LIN {X 53.277,Y 73.918,Z 73.500,A 180.000,B 0.000,C 180.000} C_DIS
LIN {X 53.455,Y 73.864,Z 73.500,A 180.000,B 0.000,C 180.000} C_DIS
LIN {X 75.444,Y 66.446,Z 73.500,A 180.000,B 0.000,C 180.000} C_DIS
LIN {X 75.534,Y 66.414,Z 73.500,A 180.000,B 0.000,C 180.000} C_DIS
LIN {X 75.623,Y 66.379,Z 73.500,A 180.000,B 0.000,C 180.000} C_DIS
LIN {X 75.739,Y 66.327,Z 73.500,A 180.000,B 0.000,C 180.000} C_DIS
LIN {X 75.802,Y 66.296,Z 73.500,A 180.000,B 0.000,C 180.000} C_DIS
LIN {X 75.891,Y 66.247,Z 73.500,A 180.000,B 0.000,C 180.000} C_DIS
LIN {X 75.980,Y 66.194,Z 73.500,A 180.000,B 0.000,C 180.000} C_DIS
LIN {X 76.052,Y 66.148,Z 73.500,A 180.000,B 0.000,C 180.000} C_DIS
LIN {X 76.159,Y 66.072,Z 73.500,A 180.000,B 0.000,C 180.000} C_DIS
LIN {X 76.223,Y 66.022,Z 73.500,A 180.000,B 0.000,C 180.000} C_DIS
LIN {X 76.287,Y 65.969,Z 73.500,A 180.000,B 0.000,C 180.000} C_DIS
LIN {X 76.338,Y 65.924,Z 73.500,A 180.000,B 0.000,C 180.000} C_DIS
LIN {X 76.406,Y 65.860,Z 73.500,A 180.000,B 0.000,C 180.000} C_DIS
LIN {X 76.474,Y 65.791,Z 73.500,A 180.000,B 0.000,C 180.000} C_DIS
LIN {X 76.517,Y 65.744,Z 73.500,A 180.000,B 0.000,C 180.000} C_DIS
LIN {X 76.628,Y 65.612,Z 73.500,A 180.000,B 0.000,C 180.000} C_DIS
LIN {X 76.696,Y 65.521,Z 73.500,A 180.000,B 0.000,C 180.000} C_DIS
LIN {X 76.755,Y 65.433,Z 73.500,A 180.000,B 0.000,C 180.000} C_DIS
LIN {X 76.861,Y 65.254,Z 73.500,A 180.000,B 0.000,C 180.000} C_DIS
LIN {X 76.874,Y 65.229,Z 73.500,A 180.000,B 0.000,C 180.000} C_DIS
LIN {X 76.948,Y 65.075,Z 73.500,A 180.000,B 0.000,C 180.000} C_DIS
LIN {X 77.018,Y 64.897,Z 73.500,A 180.000,B 0.000,C 180.000} C_DIS
LIN {X 77.053,Y 64.789,Z 73.500,A 180.000,B 0.000,C 180.000} C_DIS
LIN {X 77.073,Y 64.718,Z 73.500,A 180.000,B 0.000,C 180.000} C_DIS
LIN {X 77.114,Y 64.539,Z 73.500,A 180.000,B 0.000,C 180.000} C_DIS
LIN {X 77.141,Y 64.360,Z 73.500,A 180.000,B 0.000,C 180.000} C_DIS
LIN {X 77.155,Y 64.182,Z 73.500,A 180.000,B 0.000,C 180.000} C_DIS
LIN {X 77.157,Y 64.003,Z 73.500,A 180.000,B 0.000,C 180.000} C_DIS
LIN {X 77.145,Y 63.824,Z 73.500,A 180.000,B 0.000,C 180.000} C_DIS
LIN {X 77.121,Y 63.645,Z 73.500,A 180.000,B 0.000,C 180.000} C_DIS
LIN {X 77.083,Y 63.467,Z 73.500,A 180.000,B 0.000,C 180.000} C_DIS
LIN {X 77.053,Y 63.357,Z 73.500,A 180.000,B 0.000,C 180.000} C_DIS
LIN {X 77.031,Y 63.288,Z 73.500,A 180.000,B 0.000,C 180.000} C_DIS
LIN {X 76.971,Y 63.109,Z 73.500,A 180.000,B 0.000,C 180.000} C_DIS
LIN {X 70.639,Y 44.338,Z 73.500,A 180.000,B 0.000,C 180.000} C_DIS
LIN {X 70.617,Y 44.276,Z 73.500,A 180.000,B 0.000,C 180.000} C_DIS
LIN {X 70.572,Y 44.159,Z 73.500,A 180.000,B 0.000,C 180.000} C_DIS
LIN {X 70.489,Y 43.981,Z 73.500,A 180.000,B 0.000,C 180.000} C_DIS
LIN {X 70.439,Y 43.887,Z 73.500,A 180.000,B 0.000,C 180.000} C_DIS
LIN {X 70.388,Y 43.802,Z 73.500,A 180.000,B 0.000,C 180.000} C_DIS
LIN {X 70.266,Y 43.623,Z 73.500,A 180.000,B 0.000,C 180.000} C_DIS
LIN {X 70.260,Y 43.615,Z 73.500,A 180.000,B 0.000,C 180.000} C_DIS
LIN {X 70.118,Y 43.444,Z 73.500,A 180.000,B 0.000,C 180.000} C_DIS
LIN {X 70.081,Y 43.404,Z 73.500,A 180.000,B 0.000,C 180.000} C_DIS
LIN {X 69.939,Y 43.266,Z 73.500,A 180.000,B 0.000,C 180.000} C_DIS
LIN {X 69.902,Y 43.233,Z 73.500,A 180.000,B 0.000,C 180.000} C_DIS
LIN {X 69.724,Y 43.092,Z 73.500,A 180.000,B 0.000,C 180.000} C_DIS
LIN {X 69.717,Y 43.087,Z 73.500,A 180.000,B 0.000,C 180.000} C_DIS
LIN {X 69.545,Y 42.975,Z 73.500,A 180.000,B 0.000,C 180.000} C_DIS
LIN {X 69.426,Y 42.908,Z 73.500,A 180.000,B 0.000,C 180.000} C_DIS
LIN {X 69.366,Y 42.878,Z 73.500,A 180.000,B 0.000,C 180.000} C_DIS
LIN {X 69.187,Y 42.798,Z 73.500,A 180.000,B 0.000,C 180.000} C_DIS
LIN {X 69.008,Y 42.735,Z 73.500,A 180.000,B 0.000,C 180.000} C_DIS
LIN {X 68.989,Y 42.729,Z 73.500,A 180.000,B 0.000,C 180.000} C_DIS
LIN {X 68.830,Y 42.687,Z 73.500,A 180.000,B 0.000,C 180.000} C_DIS
LIN {X 68.651,Y 42.652,Z 73.500,A 180.000,B 0.000,C 180.000} C_DIS
LIN {X 68.562,Y 42.640,Z 73.500,A 180.000,B 0.000,C 180.000} C_DIS
LIN {X 68.472,Y 42.631,Z 73.500,A 180.000,B 0.000,C 180.000} C_DIS
LIN {X 68.383,Y 42.625,Z 73.500,A 180.000,B 0.000,C 180.000} C_DIS
LIN {X 68.293,Y 42.622,Z 73.500,A 180.000,B 0.000,C 180.000} C_DIS
LIN {X 68.204,Y 42.623,Z 73.500,A 180.000,B 0.000,C 180.000} C_DIS
LIN {X 68.115,Y 42.627,Z 73.500,A 180.000,B 0.000,C 180.000} C_DIS
LIN {X 68.025,Y 42.634,Z 73.500,A 180.000,B 0.000,C 180.000} C_DIS
LIN {X 67.936,Y 42.644,Z 73.500,A 180.000,B 0.000,C 180.000} C_DIS
LIN {X 67.846,Y 42.657,Z 73.500,A 180.000,B 0.000,C 180.000} C_DIS
LIN {X 67.757,Y 42.674,Z 73.500,A 180.000,B 0.000,C 180.000} C_DIS
LIN {X 67.668,Y 42.694,Z 73.500,A 180.000,B 0.000,C 180.000} C_DIS
LIN {X 67.578,Y 42.718,Z 73.500,A 180.000,B 0.000,C 180.000} C_DIS
LIN {X 67.541,Y 42.729,Z 73.500,A 180.000,B 0.000,C 180.000} C_DIS
LIN {X 67.399,Y 42.776,Z 73.500,A 180.000,B 0.000,C 180.000} C_DIS
LIN {X 47.482,Y 49.495,Z 73.500,A 180.000,B 0.000,C 180.000} C_DIS
; Link Move Starts
LIN {X 47.184,Y 49.595,Z 73.500,A 180.000,B 0.000,C 180.000} C_DIS
LIN {X 46.885,Y 49.696,Z 73.499,A 180.000,B 0.000,C 180.000} C_DIS
LIN {X 46.587,Y 49.797,Z 73.498,A 180.000,B 0.000,C 180.000} C_DIS
LIN {X 46.288,Y 49.897,Z 73.496,A 180.000,B 0.000,C 180.000} C_DIS
LIN {X 45.990,Y 49.998,Z 73.494,A 180.000,B 0.000,C 180.000} C_DIS
LIN {X 45.692,Y 50.099,Z 73.491,A 180.000,B 0.000,C 180.000} C_DIS
LIN {X 45.393,Y 50.200,Z 73.488,A 180.000,B 0.000,C 180.000} C_DIS
LIN {X 45.247,Y 50.259,Z 73.487,A 180.000,B 0.000,C 180.000} C_DIS
LIN {X 45.105,Y 50.326,Z 73.485,A 180.000,B 0.000,C 180.000} C_DIS
LIN {X 44.967,Y 50.403,Z 73.483,A 180.000,B 0.000,C 180.000} C_DIS
LIN {X 44.834,Y 50.487,Z 73.481,A 180.000,B 0.000,C 180.000} C_DIS
LIN {X 44.707,Y 50.581,Z 73.479,A 180.000,B 0.000,C 180.000} C_DIS
LIN {X 44.587,Y 50.682,Z 73.477,A 180.000,B 0.000,C 180.000} C_DIS
LIN {X 44.472,Y 50.790,Z 73.474,A 180.000,B 0.000,C 180.000} C_DIS
LIN {X 44.365,Y 50.905,Z 73.472,A 180.000,B 0.000,C 180.000} C_DIS
LIN {X 44.265,Y 51.027,Z 73.469,A 180.000,B 0.000,C 180.000} C_DIS
LIN {X 44.173,Y 51.155,Z 73.467,A 180.000,B 0.000,C 180.000} C_DIS
LIN {X 44.090,Y 51.288,Z 73.464,A 180.000,B 0.000,C 180.000} C_DIS
LIN {X 44.014,Y 51.427,Z 73.461,A 180.000,B 0.000,C 180.000} C_DIS
LIN {X 43.948,Y 51.570,Z 73.459,A 180.000,B 0.000,C 180.000} C_DIS
LIN {X 43.891,Y 51.716,Z 73.456,A 180.000,B 0.000,C 180.000} C_DIS
LIN {X 43.843,Y 51.867,Z 73.452,A 180.000,B 0.000,C 180.000} C_DIS
LIN {X 43.805,Y 52.019,Z 73.449,A 180.000,B 0.000,C 180.000} C_DIS
LIN {X 43.777,Y 52.174,Z 73.446,A 180.000,B 0.000,C 180.000} C_DIS
LIN {X 43.758,Y 52.331,Z 73.443,A 180.000,B 0.000,C 180.000} C_DIS
LIN {X 43.749,Y 52.488,Z 73.439,A 180.000,B 0.000,C 180.000} C_DIS
LIN {X 43.750,Y 52.645,Z 73.436,A 180.000,B 0.000,C 180.000} C_DIS
LIN {X 43.761,Y 52.803,Z 73.432,A 180.000,B 0.000,C 180.000} C_DIS
LIN {X 43.782,Y 52.959,Z 73.428,A 180.000,B 0.000,C 180.000} C_DIS
LIN {X 43.813,Y 53.113,Z 73.425,A 180.000,B 0.000,C 180.000} C_DIS
LIN {X 43.853,Y 53.265,Z 73.421,A 180.000,B 0.000,C 180.000} C_DIS
LIN {X 43.902,Y 53.415,Z 73.417,A 180.000,B 0.000,C 180.000} C_DIS
LIN {X 43.952,Y 53.564,Z 73.413,A 180.000,B 0.000,C 180.000} C_DIS
LIN {X 44.003,Y 53.714,Z 73.409,A 180.000,B 0.000,C 180.000} C_DIS
LIN {X 44.053,Y 53.863,Z 73.405,A 180.000,B 0.000,C 180.000} C_DIS
LIN {X 44.103,Y 54.012,Z 73.400,A 180.000,B 0.000,C 180.000} C_DIS
LIN {X 44.154,Y 54.161,Z 73.396,A 180.000,B 0.000,C 180.000} C_DIS
LIN {X 44.204,Y 54.310,Z 73.392,A 180.000,B 0.000,C 180.000} C_DIS
LIN {X 44.254,Y 54.460,Z 73.387,A 180.000,B 0.000,C 180.000} C_DIS
LIN {X 44.305,Y 54.609,Z 73.383,A 180.000,B 0.000,C 180.000} C_DIS
LIN {X 44.355,Y 54.758,Z 73.378,A 180.000,B 0.000,C 180.000} C_DIS
LIN {X 44.405,Y 54.907,Z 73.373,A 180.000,B 0.000,C 180.000} C_DIS
LIN {X 44.456,Y 55.057,Z 73.369,A 180.000,B 0.000,C 180.000} C_DIS
LIN {X 44.506,Y 55.206,Z 73.364,A 180.000,B 0.000,C 180.000} C_DIS
LIN {X 44.556,Y 55.355,Z 73.359,A 180.000,B 0.000,C 180.000} C_DIS
LIN {X 44.607,Y 55.504,Z 73.354,A 180.000,B 0.000,C 180.000} C_DIS
LIN {X 44.632,Y 55.579,Z 73.351,A 180.000,B 0.000,C 180.000} C_DIS
LIN {X 44.657,Y 55.654,Z 73.349,A 180.000,B 0.000,C 180.000} C_DIS
LIN {X 44.682,Y 55.728,Z 73.346,A 180.000,B 0.000,C 180.000} C_DIS
LIN {X 44.707,Y 55.803,Z 73.344,A 180.000,B 0.000,C 180.000} C_DIS
LIN {X 44.733,Y 55.877,Z 73.341,A 180.000,B 0.000,C 180.000} C_DIS
LIN {X 44.758,Y 55.952,Z 73.339,A 180.000,B 0.000,C 180.000} C_DIS
LIN {X 44.783,Y 56.027,Z 73.336,A 180.000,B 0.000,C 180.000} C_DIS
LIN {X 44.833,Y 56.176,Z 73.331,A 180.000,B 0.000,C 180.000} C_DIS
LIN {X 44.884,Y 56.325,Z 73.325,A 180.000,B 0.000,C 180.000} C_DIS
LIN {X 44.934,Y 56.474,Z 73.320,A 180.000,B 0.000,C 180.000} C_DIS
LIN {X 44.984,Y 56.624,Z 73.315,A 180.000,B 0.000,C 180.000} C_DIS
LIN {X 45.035,Y 56.773,Z 73.309,A 180.000,B 0.000,C 180.000} C_DIS
LIN {X 45.060,Y 56.848,Z 73.307,A 180.000,B 0.000,C 180.000} C_DIS
LIN {X 45.110,Y 56.997,Z 73.301,A 180.000,B 0.000,C 180.000} C_DIS
LIN {X 45.186,Y 57.221,Z 73.293,A 180.000,B 0.000,C 180.000} C_DIS
LIN {X 45.236,Y 57.370,Z 73.287,A 180.000,B 0.000,C 180.000} C_DIS
LIN {X 45.261,Y 57.444,Z 73.285,A 180.000,B 0.000,C 180.000} C_DIS
LIN {X 45.312,Y 57.594,Z 73.279,A 180.000,B 0.000,C 180.000} C_DIS
LIN {X 45.387,Y 57.818,Z 73.271,A 180.000,B 0.000,C 180.000} C_DIS
LIN {X 45.437,Y 57.967,Z 73.265,A 180.000,B 0.000,C 180.000} C_DIS
LIN {X 45.463,Y 58.041,Z 73.263,A 180.000,B 0.000,C 180.000} C_DIS
LIN {X 45.513,Y 58.191,Z 73.257,A 180.000,B 0.000,C 180.000} C_DIS
LIN {X 45.588,Y 58.414,Z 73.249,A 180.000,B 0.000,C 180.000} C_DIS
LIN {X 45.639,Y 58.564,Z 73.243,A 180.000,B 0.000,C 180.000} C_DIS
LIN {X 45.664,Y 58.638,Z 73.241,A 180.000,B 0.000,C 180.000} C_DIS
LIN {X 45.714,Y 58.788,Z 73.235,A 180.000,B 0.000,C 180.000} C_DIS
LIN {X 45.790,Y 59.011,Z 73.227,A 180.000,B 0.000,C 180.000} C_DIS
LIN {X 45.840,Y 59.161,Z 73.221,A 180.000,B 0.000,C 180.000} C_DIS
LIN {X 45.865,Y 59.235,Z 73.219,A 180.000,B 0.000,C 180.000} C_DIS
LIN {X 45.916,Y 59.385,Z 73.213,A 180.000,B 0.000,C 180.000} C_DIS
LIN {X 46.067,Y 59.832,Z 73.197,A 180.000,B 0.000,C 180.000} C_DIS
LIN {X 46.117,Y 59.981,Z 73.191,A 180.000,B 0.000,C 180.000} C_DIS
LIN {X 46.268,Y 60.429,Z 73.175,A 180.000,B 0.000,C 180.000} C_DIS
LIN {X 46.318,Y 60.578,Z 73.169,A 180.000,B 0.000,C 180.000} C_DIS
LIN {X 46.495,Y 61.101,Z 73.150,A 180.000,B 0.000,C 180.000} C_DIS
LIN {X 46.646,Y 61.548,Z 73.133,A 180.000,B 0.000,C 180.000} C_DIS
LIN {X 46.696,Y 61.698,Z 73.128,A 180.000,B 0.000,C 180.000} C_DIS
LIN {X 46.847,Y 62.145,Z 73.111,A 180.000,B 0.000,C 180.000} C_DIS
LIN {X 46.897,Y 62.295,Z 73.106,A 180.000,B 0.000,C 180.000} C_DIS
LIN {X 47.149,Y 63.041,Z 73.078,A 180.000,B 0.000,C 180.000} C_DIS
LIN {X 47.275,Y 63.414,Z 73.065,A 180.000,B 0.000,C 180.000} C_DIS
LIN {X 47.426,Y 63.862,Z 73.048,A 180.000,B 0.000,C 180.000} C_DIS
LIN {X 48.005,Y 65.578,Z 72.985,A 180.000,B 0.000,C 180.000} C_DIS
LIN {X 48.962,Y 68.413,Z 72.880,A 180.000,B 0.000,C 180.000} C_DIS
LIN {X 49.012,Y 68.563,Z 72.875,A 180.000,B 0.000,C 180.000} C_DIS
LIN {X 49.163,Y 69.010,Z 72.858,A 180.000,B 0.000,C 180.000} C_DIS
LIN {X 49.213,Y 69.160,Z 72.853,A 180.000,B 0.000,C 180.000} C_DIS
LIN {X 49.364,Y 69.607,Z 72.836,A 180.000,B 0.000,C 180.000} C_DIS
LIN {X 49.390,Y 69.682,Z 72.834,A 180.000,B 0.000,C 180.000} C_DIS
LIN {X 49.440,Y 69.831,Z 72.828,A 180.000,B 0.000,C 180.000} C_DIS
LIN {X 49.591,Y 70.279,Z 72.812,A 180.000,B 0.000,C 180.000} C_DIS
LIN {X 49.641,Y 70.428,Z 72.806,A 180.000,B 0.000,C 180.000} C_DIS
LIN {X 49.792,Y 70.876,Z 72.790,A 180.000,B 0.000,C 180.000} C_DIS
LIN {X 49.843,Y 71.025,Z 72.784,A 180.000,B 0.000,C 180.000} C_DIS
LIN {X 49.918,Y 71.249,Z 72.776,A 180.000,B 0.000,C 180.000} C_DIS
LIN {X 49.968,Y 71.398,Z 72.770,A 180.000,B 0.000,C 180.000} C_DIS
LIN {X 49.994,Y 71.473,Z 72.768,A 180.000,B 0.000,C 180.000} C_DIS
LIN {X 50.044,Y 71.622,Z 72.762,A 180.000,B 0.000,C 180.000} C_DIS
LIN {X 50.120,Y 71.846,Z 72.754,A 180.000,B 0.000,C 180.000} C_DIS
LIN {X 50.170,Y 71.995,Z 72.748,A 180.000,B 0.000,C 180.000} C_DIS
LIN {X 50.195,Y 72.070,Z 72.746,A 180.000,B 0.000,C 180.000} C_DIS
LIN {X 50.245,Y 72.219,Z 72.740,A 180.000,B 0.000,C 180.000} C_DIS
LIN {X 50.271,Y 72.293,Z 72.737,A 180.000,B 0.000,C 180.000} C_DIS
LIN {X 50.297,Y 72.368,Z 72.735,A 180.000,B 0.000,C 180.000} C_DIS
LIN {X 50.325,Y 72.441,Z 72.732,A 180.000,B 0.000,C 180.000} C_DIS
LIN {X 50.356,Y 72.514,Z 72.729,A 180.000,B 0.000,C 180.000} C_DIS
LIN {X 50.389,Y 72.585,Z 72.726,A 180.000,B 0.000,C 180.000} C_DIS
LIN {X 50.424,Y 72.656,Z 72.724,A 180.000,B 0.000,C 180.000} C_DIS
LIN {X 50.462,Y 72.725,Z 72.721,A 180.000,B 0.000,C 180.000} C_DIS
LIN {X 50.502,Y 72.793,Z 72.718,A 180.000,B 0.000,C 180.000} C_DIS
LIN {X 50.543,Y 72.860,Z 72.715,A 180.000,B 0.000,C 180.000} C_DIS
LIN {X 50.587,Y 72.925,Z 72.713,A 180.000,B 0.000,C 180.000} C_DIS
LIN {X 50.633,Y 72.989,Z 72.710,A 180.000,B 0.000,C 180.000} C_DIS
LIN {X 50.681,Y 73.052,Z 72.707,A 180.000,B 0.000,C 180.000} C_DIS
LIN {X 50.731,Y 73.113,Z 72.704,A 180.000,B 0.000,C 180.000} C_DIS
LIN {X 50.783,Y 73.172,Z 72.702,A 180.000,B 0.000,C 180.000} C_DIS
LIN {X 50.836,Y 73.230,Z 72.699,A 180.000,B 0.000,C 180.000} C_DIS
LIN {X 50.892,Y 73.286,Z 72.696,A 180.000,B 0.000,C 180.000} C_DIS
LIN {X 50.949,Y 73.340,Z 72.693,A 180.000,B 0.000,C 180.000} C_DIS
LIN {X 51.008,Y 73.392,Z 72.691,A 180.000,B 0.000,C 180.000} C_DIS
LIN {X 51.068,Y 73.443,Z 72.688,A 180.000,B 0.000,C 180.000} C_DIS
LIN {X 51.130,Y 73.491,Z 72.685,A 180.000,B 0.000,C 180.000} C_DIS
LIN {X 51.193,Y 73.538,Z 72.682,A 180.000,B 0.000,C 180.000} C_DIS
LIN {X 51.258,Y 73.583,Z 72.680,A 180.000,B 0.000,C 180.000} C_DIS
LIN {X 51.325,Y 73.625,Z 72.677,A 180.000,B 0.000,C 180.000} C_DIS
LIN {X 51.392,Y 73.666,Z 72.674,A 180.000,B 0.000,C 180.000} C_DIS
LIN {X 51.461,Y 73.704,Z 72.672,A 180.000,B 0.000,C 180.000} C_DIS
LIN {X 51.531,Y 73.740,Z 72.669,A 180.000,B 0.000,C 180.000} C_DIS
LIN {X 51.602,Y 73.774,Z 72.666,A 180.000,B 0.000,C 180.000} C_DIS
LIN {X 51.674,Y 73.805,Z 72.664,A 180.000,B 0.000,C 180.000} C_DIS
LIN {X 51.747,Y 73.835,Z 72.661,A 180.000,B 0.000,C 180.000} C_DIS
LIN {X 51.821,Y 73.862,Z 72.659,A 180.000,B 0.000,C 180.000} C_DIS
LIN {X 51.896,Y 73.886,Z 72.656,A 180.000,B 0.000,C 180.000} C_DIS
LIN {X 51.972,Y 73.909,Z 72.654,A 180.000,B 0.000,C 180.000} C_DIS
LIN {X 52.048,Y 73.929,Z 72.651,A 180.000,B 0.000,C 180.000} C_DIS
LIN {X 52.125,Y 73.946,Z 72.648,A 180.000,B 0.000,C 180.000} C_DIS
LIN {X 52.280,Y 73.974,Z 72.644,A 180.000,B 0.000,C 180.000} C_DIS
LIN {X 52.436,Y 73.992,Z 72.639,A 180.000,B 0.000,C 180.000} C_DIS
LIN {X 52.594,Y 74.000,Z 72.634,A 180.000,B 0.000,C 180.000} C_DIS
LIN {X 52.751,Y 73.998,Z 72.629,A 180.000,B 0.000,C 180.000} C_DIS
LIN {X 52.908,Y 73.986,Z 72.624,A 180.000,B 0.000,C 180.000} C_DIS
LIN {X 53.064,Y 73.964,Z 72.620,A 180.000,B 0.000,C 180.000} C_DIS
LIN {X 53.218,Y 73.932,Z 72.615,A 180.000,B 0.000,C 180.000} C_DIS
LIN {X 53.370,Y 73.891,Z 72.610,A 180.000,B 0.000,C 180.000} C_DIS
LIN {X 53.520,Y 73.842,Z 72.606,A 180.000,B 0.000,C 180.000} C_DIS
LIN {X 53.669,Y 73.792,Z 72.602,A 180.000,B 0.000,C 180.000} C_DIS
LIN {X 53.819,Y 73.741,Z 72.597,A 180.000,B 0.000,C 180.000} C_DIS
LIN {X 53.968,Y 73.691,Z 72.593,A 180.000,B 0.000,C 180.000} C_DIS
LIN {X 54.117,Y 73.641,Z 72.589,A 180.000,B 0.000,C 180.000} C_DIS
LIN {X 54.266,Y 73.590,Z 72.585,A 180.000,B 0.000,C 180.000} C_DIS
LIN {X 54.415,Y 73.540,Z 72.581,A 180.000,B 0.000,C 180.000} C_DIS
LIN {X 54.565,Y 73.490,Z 72.577,A 180.000,B 0.000,C 180.000} C_DIS
LIN {X 54.714,Y 73.439,Z 72.573,A 180.000,B 0.000,C 180.000} C_DIS
LIN {X 54.863,Y 73.389,Z 72.570,A 180.000,B 0.000,C 180.000} C_DIS
LIN {X 55.012,Y 73.339,Z 72.566,A 180.000,B 0.000,C 180.000} C_DIS
LIN {X 55.162,Y 73.288,Z 72.562,A 180.000,B 0.000,C 180.000} C_DIS
LIN {X 55.311,Y 73.238,Z 72.559,A 180.000,B 0.000,C 180.000} C_DIS
LIN {X 55.460,Y 73.187,Z 72.556,A 180.000,B 0.000,C 180.000} C_DIS
LIN {X 55.609,Y 73.137,Z 72.552,A 180.000,B 0.000,C 180.000} C_DIS
LIN {X 55.759,Y 73.087,Z 72.549,A 180.000,B 0.000,C 180.000} C_DIS
LIN {X 55.908,Y 73.036,Z 72.546,A 180.000,B 0.000,C 180.000} C_DIS
LIN {X 56.057,Y 72.986,Z 72.543,A 180.000,B 0.000,C 180.000} C_DIS
LIN {X 56.206,Y 72.936,Z 72.540,A 180.000,B 0.000,C 180.000} C_DIS
LIN {X 56.356,Y 72.885,Z 72.537,A 180.000,B 0.000,C 180.000} C_DIS
LIN {X 56.505,Y 72.835,Z 72.534,A 180.000,B 0.000,C 180.000} C_DIS
LIN {X 56.654,Y 72.785,Z 72.532,A 180.000,B 0.000,C 180.000} C_DIS
LIN {X 56.803,Y 72.734,Z 72.529,A 180.000,B 0.000,C 180.000} C_DIS
LIN {X 56.953,Y 72.684,Z 72.527,A 180.000,B 0.000,C 180.000} C_DIS
LIN {X 57.251,Y 72.583,Z 72.522,A 180.000,B 0.000,C 180.000} C_DIS
LIN {X 57.549,Y 72.483,Z 72.518,A 180.000,B 0.000,C 180.000} C_DIS
LIN {X 57.848,Y 72.382,Z 72.514,A 180.000,B 0.000,C 180.000} C_DIS
LIN {X 58.146,Y 72.281,Z 72.511,A 180.000,B 0.000,C 180.000} C_DIS
LIN {X 58.445,Y 72.181,Z 72.508,A 180.000,B 0.000,C 180.000} C_DIS
LIN {X 58.743,Y 72.080,Z 72.505,A 180.000,B 0.000,C 180.000} C_DIS
LIN {X 59.042,Y 71.979,Z 72.503,A 180.000,B 0.000,C 180.000} C_DIS
LIN {X 59.340,Y 71.879,Z 72.502,A 180.000,B 0.000,C 180.000} C_DIS
LIN {X 59.639,Y 71.778,Z 72.501,A 180.000,B 0.000,C 180.000} C_DIS
LIN {X 59.937,Y 71.677,Z 72.500,A 180.000,B 0.000,C 180.000} C_DIS
LIN {X 60.157,Y 71.603,Z 72.500,A 180.000,B 0.000,C 180.000} C_DIS
; Cutting Move Starts
LIN {X 76.696,Y 66.024,Z 72.500,A 180.000,B 0.000,C 180.000} C_DIS
LIN {X 76.851,Y 65.969,Z 72.500,A 180.000,B 0.000,C 180.000} C_DIS
LIN {X 76.874,Y 65.961,Z 72.500,A 180.000,B 0.000,C 180.000} C_DIS
LIN {X 76.964,Y 65.924,Z 72.500,A 180.000,B 0.000,C 180.000} C_DIS
LIN {X 77.053,Y 65.883,Z 72.500,A 180.000,B 0.000,C 180.000} C_DIS
LIN {X 77.140,Y 65.839,Z 72.500,A 180.000,B 0.000,C 180.000} C_DIS
LIN {X 77.226,Y 65.791,Z 72.500,A 180.000,B 0.000,C 180.000} C_DIS
LIN {X 77.232,Y 65.787,Z 72.500,A 180.000,B 0.000,C 180.000} C_DIS
LIN {X 77.321,Y 65.732,Z 72.500,A 180.000,B 0.000,C 180.000} C_DIS
LIN {X 77.411,Y 65.672,Z 72.500,A 180.000,B 0.000,C 180.000} C_DIS
LIN {X 77.492,Y 65.612,Z 72.500,A 180.000,B 0.000,C 180.000} C_DIS
LIN {X 77.589,Y 65.532,Z 72.500,A 180.000,B 0.000,C 180.000} C_DIS
LIN {X 77.699,Y 65.433,Z 72.500,A 180.000,B 0.000,C 180.000} C_DIS
LIN {X 77.768,Y 65.364,Z 72.500,A 180.000,B 0.000,C 180.000} C_DIS
LIN {X 77.867,Y 65.254,Z 72.500,A 180.000,B 0.000,C 180.000} C_DIS
LIN {X 77.947,Y 65.156,Z 72.500,A 180.000,B 0.000,C 180.000} C_DIS
LIN {X 78.006,Y 65.075,Z 72.500,A 180.000,B 0.000,C 180.000} C_DIS
LIN {X 78.122,Y 64.897,Z 72.500,A 180.000,B 0.000,C 180.000} C_DIS
LIN {X 78.126,Y 64.890,Z 72.500,A 180.000,B 0.000,C 180.000} C_DIS
LIN {X 78.217,Y 64.718,Z 72.500,A 180.000,B 0.000,C 180.000} C_DIS
LIN {X 78.295,Y 64.539,Z 72.500,A 180.000,B 0.000,C 180.000} C_DIS
LIN {X 78.304,Y 64.514,Z 72.500,A 180.000,B 0.000,C 180.000} C_DIS
LIN {X 78.357,Y 64.360,Z 72.500,A 180.000,B 0.000,C 180.000} C_DIS
LIN {X 78.404,Y 64.182,Z 72.500,A 180.000,B 0.000,C 180.000} C_DIS
LIN {X 78.438,Y 64.003,Z 72.500,A 180.000,B 0.000,C 180.000} C_DIS
LIN {X 78.458,Y 63.824,Z 72.500,A 180.000,B 0.000,C 180.000} C_DIS
LIN {X 78.465,Y 63.645,Z 72.500,A 180.000,B 0.000,C 180.000} C_DIS
LIN {X 78.460,Y 63.467,Z 72.500,A 180.000,B 0.000,C 180.000} C_DIS
LIN {X 78.442,Y 63.288,Z 72.500,A 180.000,B 0.000,C 180.000} C_DIS
LIN {X 78.410,Y 63.109,Z 72.500,A 180.000,B 0.000,C 180.000} C_DIS
LIN {X 78.365,Y 62.930,Z 72.500,A 180.000,B 0.000,C 180.000} C_DIS
LIN {X 78.307,Y 62.751,Z 72.500,A 180.000,B 0.000,C 180.000} C_DIS
LIN {X 71.975,Y 43.981,Z 72.500,A 180.000,B 0.000,C 180.000} C_DIS
LIN {X 71.913,Y 43.802,Z 72.500,A 180.000,B 0.000,C 180.000} C_DIS
LIN {X 71.869,Y 43.692,Z 72.500,A 180.000,B 0.000,C 180.000} C_DIS
LIN {X 71.838,Y 43.623,Z 72.500,A 180.000,B 0.000,C 180.000} C_DIS
LIN {X 71.745,Y 43.444,Z 72.500,A 180.000,B 0.000,C 180.000} C_DIS
LIN {X 71.690,Y 43.352,Z 72.500,A 180.000,B 0.000,C 180.000} C_DIS
LIN {X 71.633,Y 43.266,Z 72.500,A 180.000,B 0.000,C 180.000} C_DIS
LIN {X 71.511,Y 43.103,Z 72.500,A 180.000,B 0.000,C 180.000} C_DIS
LIN {X 71.498,Y 43.087,Z 72.500,A 180.000,B 0.000,C 180.000} C_DIS
LIN {X 71.335,Y 42.908,Z 72.500,A 180.000,B 0.000,C 180.000} C_DIS
LIN {X 71.332,Y 42.905,Z 72.500,A 180.000,B 0.000,C 180.000} C_DIS
LIN {X 71.154,Y 42.744,Z 72.500,A 180.000,B 0.000,C 180.000} C_DIS
LIN {X 71.135,Y 42.729,Z 72.500,A 180.000,B 0.000,C 180.000} C_DIS
LIN {X 70.975,Y 42.611,Z 72.500,A 180.000,B 0.000,C 180.000} C_DIS
LIN {X 70.881,Y 42.550,Z 72.500,A 180.000,B 0.000,C 180.000} C_DIS
LIN {X 70.796,Y 42.501,Z 72.500,A 180.000,B 0.000,C 180.000} C_DIS
LIN {X 70.617,Y 42.410,Z 72.500,A 180.000,B 0.000,C 180.000} C_DIS
LIN {X 70.530,Y 42.372,Z 72.500,A 180.000,B 0.000,C 180.000} C_DIS
LIN {X 70.439,Y 42.336,Z 72.500,A 180.000,B 0.000,C 180.000} C_DIS
LIN {X 70.260,Y 42.277,Z 72.500,A 180.000,B 0.000,C 180.000} C_DIS
LIN {X 70.081,Y 42.233,Z 72.500,A 180.000,B 0.000,C 180.000} C_DIS
LIN {X 69.902,Y 42.203,Z 72.500,A 180.000,B 0.000,C 180.000} C_DIS
LIN {X 69.817,Y 42.193,Z 72.500,A 180.000,B 0.000,C 180.000} C_DIS
LIN {X 69.724,Y 42.185,Z 72.500,A 180.000,B 0.000,C 180.000} C_DIS
LIN {X 69.634,Y 42.182,Z 72.500,A 180.000,B 0.000,C 180.000} C_DIS
LIN {X 69.545,Y 42.181,Z 72.500,A 180.000,B 0.000,C 180.000} C_DIS
LIN {X 69.455,Y 42.184,Z 72.500,A 180.000,B 0.000,C 180.000} C_DIS
LIN {X 69.366,Y 42.189,Z 72.500,A 180.000,B 0.000,C 180.000} C_DIS
LIN {X 69.327,Y 42.193,Z 72.500,A 180.000,B 0.000,C 180.000} C_DIS
LIN {X 69.257,Y 42.201,Z 72.500,A 180.000,B 0.000,C 180.000} C_DIS
LIN {X 69.187,Y 42.211,Z 72.500,A 180.000,B 0.000,C 180.000} C_DIS
LIN {X 69.098,Y 42.226,Z 72.500,A 180.000,B 0.000,C 180.000} C_DIS
LIN {X 69.008,Y 42.245,Z 72.500,A 180.000,B 0.000,C 180.000} C_DIS
LIN {X 68.919,Y 42.268,Z 72.500,A 180.000,B 0.000,C 180.000} C_DIS
LIN {X 68.830,Y 42.294,Z 72.500,A 180.000,B 0.000,C 180.000} C_DIS
LIN {X 68.651,Y 42.353,Z 72.500,A 180.000,B 0.000,C 180.000} C_DIS
LIN {X 47.482,Y 49.495,Z 72.500,A 180.000,B 0.000,C 180.000} C_DIS
LIN {X 45.590,Y 50.133,Z 72.500,A 180.000,B 0.000,C 180.000} C_DIS
LIN {X 45.411,Y 50.194,Z 72.500,A 180.000,B 0.000,C 180.000} C_DIS
LIN {X 45.296,Y 50.238,Z 72.500,A 180.000,B 0.000,C 180.000} C_DIS
LIN {X 45.232,Y 50.265,Z 72.500,A 180.000,B 0.000,C 180.000} C_DIS
LIN {X 45.053,Y 50.353,Z 72.500,A 180.000,B 0.000,C 180.000} C_DIS
LIN {X 44.944,Y 50.416,Z 72.500,A 180.000,B 0.000,C 180.000} C_DIS
LIN {X 44.874,Y 50.461,Z 72.500,A 180.000,B 0.000,C 180.000} C_DIS
LIN {X 44.785,Y 50.522,Z 72.500,A 180.000,B 0.000,C 180.000} C_DIS
LIN {X 44.696,Y 50.590,Z 72.500,A 180.000,B 0.000,C 180.000} C_DIS
LIN {X 44.689,Y 50.595,Z 72.500,A 180.000,B 0.000,C 180.000} C_DIS
LIN {X 44.603,Y 50.667,Z 72.500,A 180.000,B 0.000,C 180.000} C_DIS
LIN {X 44.517,Y 50.746,Z 72.500,A 180.000,B 0.000,C 180.000} C_DIS
LIN {X 44.488,Y 50.774,Z 72.500,A 180.000,B 0.000,C 180.000} C_DIS
LIN {X 44.410,Y 50.855,Z 72.500,A 180.000,B 0.000,C 180.000} C_DIS
LIN {X 44.338,Y 50.936,Z 72.500,A 180.000,B 0.000,C 180.000} C_DIS
LIN {X 44.325,Y 50.953,Z 72.500,A 180.000,B 0.000,C 180.000} C_DIS
LIN {X 44.254,Y 51.042,Z 72.500,A 180.000,B 0.000,C 180.000} C_DIS
LIN {X 44.189,Y 51.131,Z 72.500,A 180.000,B 0.000,C 180.000} C_DIS
LIN {X 44.159,Y 51.176,Z 72.500,A 180.000,B 0.000,C 180.000} C_DIS
LIN {X 44.077,Y 51.310,Z 72.500,A 180.000,B 0.000,C 180.000} C_DIS
LIN {X 43.984,Y 51.489,Z 72.500,A 180.000,B 0.000,C 180.000} C_DIS
LIN {X 43.981,Y 51.497,Z 72.500,A 180.000,B 0.000,C 180.000} C_DIS
LIN {X 43.909,Y 51.668,Z 72.500,A 180.000,B 0.000,C 180.000} C_DIS
LIN {X 43.849,Y 51.847,Z 72.500,A 180.000,B 0.000,C 180.000} C_DIS
LIN {X 43.804,Y 52.025,Z 72.500,A 180.000,B 0.000,C 180.000} C_DIS
LIN {X 43.802,Y 52.035,Z 72.500,A 180.000,B 0.000,C 180.000} C_DIS
LIN {X 43.772,Y 52.204,Z 72.500,A 180.000,B 0.000,C 180.000} C_DIS
LIN {X 43.754,Y 52.383,Z 72.500,A 180.000,B 0.000,C 180.000} C_DIS
LIN {X 43.748,Y 52.562,Z 72.500,A 180.000,B 0.000,C 180.000} C_DIS
LIN {X 43.756,Y 52.740,Z 72.500,A 180.000,B 0.000,C 180.000} C_DIS
LIN {X 43.776,Y 52.919,Z 72.500,A 180.000,B 0.000,C 180.000} C_DIS
LIN {X 43.802,Y 53.064,Z 72.500,A 180.000,B 0.000,C 180.000} C_DIS
LIN {X 43.809,Y 53.098,Z 72.500,A 180.000,B 0.000,C 180.000} C_DIS
LIN {X 43.856,Y 53.277,Z 72.500,A 180.000,B 0.000,C 180.000} C_DIS
LIN {X 43.916,Y 53.455,Z 72.500,A 180.000,B 0.000,C 180.000} C_DIS
LIN {X 50.248,Y 72.226,Z 72.500,A 180.000,B 0.000,C 180.000} C_DIS
LIN {X 50.311,Y 72.405,Z 72.500,A 180.000,B 0.000,C 180.000} C_DIS
LIN {X 50.388,Y 72.584,Z 72.500,A 180.000,B 0.000,C 180.000} C_DIS
LIN {X 50.416,Y 72.640,Z 72.500,A 180.000,B 0.000,C 180.000} C_DIS
LIN {X 50.484,Y 72.763,Z 72.500,A 180.000,B 0.000,C 180.000} C_DIS
LIN {X 50.595,Y 72.936,Z 72.500,A 180.000,B 0.000,C 180.000} C_DIS
LIN {X 50.599,Y 72.941,Z 72.500,A 180.000,B 0.000,C 180.000} C_DIS
LIN {X 50.665,Y 73.031,Z 72.500,A 180.000,B 0.000,C 180.000} C_DIS
LIN {X 50.737,Y 73.120,Z 72.500,A 180.000,B 0.000,C 180.000} C_DIS
LIN {X 50.774,Y 73.162,Z 72.500,A 180.000,B 0.000,C 180.000} C_DIS
LIN {X 50.905,Y 73.299,Z 72.500,A 180.000,B 0.000,C 180.000} C_DIS
LIN {X 50.953,Y 73.343,Z 72.500,A 180.000,B 0.000,C 180.000} C_DIS
LIN {X 51.112,Y 73.478,Z 72.500,A 180.000,B 0.000,C 180.000} C_DIS
LIN {X 51.131,Y 73.493,Z 72.500,A 180.000,B 0.000,C 180.000} C_DIS
LIN {X 51.310,Y 73.616,Z 72.500,A 180.000,B 0.000,C 180.000} C_DIS
LIN {X 51.376,Y 73.656,Z 72.500,A 180.000,B 0.000,C 180.000} C_DIS
LIN {X 51.489,Y 73.719,Z 72.500,A 180.000,B 0.000,C 180.000} C_DIS
LIN {X 51.668,Y 73.803,Z 72.500,A 180.000,B 0.000,C 180.000} C_DIS
LIN {X 51.749,Y 73.835,Z 72.500,A 180.000,B 0.000,C 180.000} C_DIS
LIN {X 51.847,Y 73.870,Z 72.500,A 180.000,B 0.000,C 180.000} C_DIS
LIN {X 52.025,Y 73.923,Z 72.500,A 180.000,B 0.000,C 180.000} C_DIS
LIN {X 52.204,Y 73.961,Z 72.500,A 180.000,B 0.000,C 180.000} C_DIS
LIN {X 52.383,Y 73.987,Z 72.500,A 180.000,B 0.000,C 180.000} C_DIS
LIN {X 52.562,Y 73.999,Z 72.500,A 180.000,B 0.000,C 180.000} C_DIS
LIN {X 52.740,Y 73.998,Z 72.500,A 180.000,B 0.000,C 180.000} C_DIS
LIN {X 52.919,Y 73.985,Z 72.500,A 180.000,B 0.000,C 180.000} C_DIS
LIN {X 53.098,Y 73.958,Z 72.500,A 180.000,B 0.000,C 180.000} C_DIS
LIN {X 53.277,Y 73.918,Z 72.500,A 180.000,B 0.000,C 180.000} C_DIS
LIN {X 53.455,Y 73.864,Z 72.500,A 180.000,B 0.000,C 180.000} C_DIS
LIN {X 57.977,Y 72.338,Z 72.500,A 180.000,B 0.000,C 180.000} C_DIS
LIN {X 60.157,Y 71.603,Z 72.500,A 180.000,B 0.000,C 180.000} C_DIS
; Link Move Starts
LIN {X 60.455,Y 71.502,Z 72.500,A 180.000,B 0.000,C 180.000} C_DIS
LIN {X 60.754,Y 71.402,Z 72.499,A 180.000,B 0.000,C 180.000} C_DIS
LIN {X 61.052,Y 71.301,Z 72.498,A 180.000,B 0.000,C 180.000} C_DIS
LIN {X 61.350,Y 71.200,Z 72.496,A 180.000,B 0.000,C 180.000} C_DIS
LIN {X 61.649,Y 71.100,Z 72.494,A 180.000,B 0.000,C 180.000} C_DIS
LIN {X 61.947,Y 70.999,Z 72.491,A 180.000,B 0.000,C 180.000} C_DIS
LIN {X 62.246,Y 70.898,Z 72.488,A 180.000,B 0.000,C 180.000} C_DIS
LIN {X 62.544,Y 70.798,Z 72.485,A 180.000,B 0.000,C 180.000} C_DIS
LIN {X 62.843,Y 70.697,Z 72.481,A 180.000,B 0.000,C 180.000} C_DIS
LIN {X 63.141,Y 70.596,Z 72.477,A 180.000,B 0.000,C 180.000} C_DIS
LIN {X 63.440,Y 70.496,Z 72.472,A 180.000,B 0.000,C 180.000} C_DIS
LIN {X 63.589,Y 70.445,Z 72.469,A 180.000,B 0.000,C 180.000} C_DIS
LIN {X 63.738,Y 70.395,Z 72.467,A 180.000,B 0.000,C 180.000} C_DIS
LIN {X 63.887,Y 70.345,Z 72.464,A 180.000,B 0.000,C 180.000} C_DIS
LIN {X 64.037,Y 70.294,Z 72.461,A 180.000,B 0.000,C 180.000} C_DIS
LIN {X 64.186,Y 70.244,Z 72.459,A 180.000,B 0.000,C 180.000} C_DIS
LIN {X 64.335,Y 70.193,Z 72.456,A 180.000,B 0.000,C 180.000} C_DIS
LIN {X 64.484,Y 70.143,Z 72.452,A 180.000,B 0.000,C 180.000} C_DIS
LIN {X 64.634,Y 70.093,Z 72.449,A 180.000,B 0.000,C 180.000} C_DIS
LIN {X 64.783,Y 70.042,Z 72.446,A 180.000,B 0.000,C 180.000} C_DIS
LIN {X 64.932,Y 69.992,Z 72.443,A 180.000,B 0.000,C 180.000} C_DIS
LIN {X 65.081,Y 69.942,Z 72.439,A 180.000,B 0.000,C 180.000} C_DIS
LIN {X 65.231,Y 69.891,Z 72.436,A 180.000,B 0.000,C 180.000} C_DIS
LIN {X 65.380,Y 69.841,Z 72.432,A 180.000,B 0.000,C 180.000} C_DIS
LIN {X 65.529,Y 69.791,Z 72.428,A 180.000,B 0.000,C 180.000} C_DIS
LIN {X 65.678,Y 69.740,Z 72.425,A 180.000,B 0.000,C 180.000} C_DIS
LIN {X 65.828,Y 69.690,Z 72.421,A 180.000,B 0.000,C 180.000} C_DIS
LIN {X 65.977,Y 69.640,Z 72.417,A 180.000,B 0.000,C 180.000} C_DIS
LIN {X 66.126,Y 69.589,Z 72.413,A 180.000,B 0.000,C 180.000} C_DIS
LIN {X 66.275,Y 69.539,Z 72.409,A 180.000,B 0.000,C 180.000} C_DIS
LIN {X 66.424,Y 69.489,Z 72.405,A 180.000,B 0.000,C 180.000} C_DIS
LIN {X 66.574,Y 69.438,Z 72.400,A 180.000,B 0.000,C 180.000} C_DIS
LIN {X 66.723,Y 69.388,Z 72.396,A 180.000,B 0.000,C 180.000} C_DIS
LIN {X 66.872,Y 69.338,Z 72.392,A 180.000,B 0.000,C 180.000} C_DIS
LIN {X 67.021,Y 69.287,Z 72.387,A 180.000,B 0.000,C 180.000} C_DIS
LIN {X 67.171,Y 69.237,Z 72.383,A 180.000,B 0.000,C 180.000} C_DIS
LIN {X 67.320,Y 69.187,Z 72.378,A 180.000,B 0.000,C 180.000} C_DIS
LIN {X 67.469,Y 69.136,Z 72.373,A 180.000,B 0.000,C 180.000} C_DIS
LIN {X 67.618,Y 69.086,Z 72.369,A 180.000,B 0.000,C 180.000} C_DIS
LIN {X 67.768,Y 69.036,Z 72.364,A 180.000,B 0.000,C 180.000} C_DIS
LIN {X 67.917,Y 68.985,Z 72.359,A 180.000,B 0.000,C 180.000} C_DIS
LIN {X 68.066,Y 68.935,Z 72.354,A 180.000,B 0.000,C 180.000} C_DIS
LIN {X 68.141,Y 68.910,Z 72.351,A 180.000,B 0.000,C 180.000} C_DIS
LIN {X 68.215,Y 68.885,Z 72.349,A 180.000,B 0.000,C 180.000} C_DIS
LIN {X 68.290,Y 68.859,Z 72.346,A 180.000,B 0.000,C 180.000} C_DIS
LIN {X 68.365,Y 68.834,Z 72.344,A 180.000,B 0.000,C 180.000} C_DIS
LIN {X 68.439,Y 68.809,Z 72.341,A 180.000,B 0.000,C 180.000} C_DIS
LIN {X 68.514,Y 68.784,Z 72.339,A 180.000,B 0.000,C 180.000} C_DIS
LIN {X 68.588,Y 68.759,Z 72.336,A 180.000,B 0.000,C 180.000} C_DIS
LIN {X 68.738,Y 68.708,Z 72.331,A 180.000,B 0.000,C 180.000} C_DIS
LIN {X 68.887,Y 68.658,Z 72.325,A 180.000,B 0.000,C 180.000} C_DIS
LIN {X 69.036,Y 68.608,Z 72.320,A 180.000,B 0.000,C 180.000} C_DIS
LIN {X 69.185,Y 68.557,Z 72.315,A 180.000,B 0.000,C 180.000} C_DIS
LIN {X 69.335,Y 68.507,Z 72.309,A 180.000,B 0.000,C 180.000} C_DIS
LIN {X 69.409,Y 68.482,Z 72.307,A 180.000,B 0.000,C 180.000} C_DIS
LIN {X 69.558,Y 68.431,Z 72.301,A 180.000,B 0.000,C 180.000} C_DIS
LIN {X 69.782,Y 68.356,Z 72.293,A 180.000,B 0.000,C 180.000} C_DIS
LIN {X 69.932,Y 68.306,Z 72.287,A 180.000,B 0.000,C 180.000} C_DIS
LIN {X 70.006,Y 68.280,Z 72.285,A 180.000,B 0.000,C 180.000} C_DIS
LIN {X 70.155,Y 68.230,Z 72.279,A 180.000,B 0.000,C 180.000} C_DIS
LIN {X 70.379,Y 68.155,Z 72.271,A 180.000,B 0.000,C 180.000} C_DIS
LIN {X 70.528,Y 68.104,Z 72.265,A 180.000,B 0.000,C 180.000} C_DIS
LIN {X 70.603,Y 68.079,Z 72.263,A 180.000,B 0.000,C 180.000} C_DIS
LIN {X 70.752,Y 68.029,Z 72.257,A 180.000,B 0.000,C 180.000} C_DIS
LIN {X 70.976,Y 67.953,Z 72.249,A 180.000,B 0.000,C 180.000} C_DIS
LIN {X 71.125,Y 67.903,Z 72.243,A 180.000,B 0.000,C 180.000} C_DIS
LIN {X 71.200,Y 67.878,Z 72.241,A 180.000,B 0.000,C 180.000} C_DIS
LIN {X 71.349,Y 67.827,Z 72.235,A 180.000,B 0.000,C 180.000} C_DIS
LIN {X 71.573,Y 67.752,Z 72.227,A 180.000,B 0.000,C 180.000} C_DIS
LIN {X 71.722,Y 67.701,Z 72.221,A 180.000,B 0.000,C 180.000} C_DIS
LIN {X 71.797,Y 67.676,Z 72.219,A 180.000,B 0.000,C 180.000} C_DIS
LIN {X 71.946,Y 67.626,Z 72.213,A 180.000,B 0.000,C 180.000} C_DIS
LIN {X 72.394,Y 67.475,Z 72.197,A 180.000,B 0.000,C 180.000} C_DIS
LIN {X 72.543,Y 67.425,Z 72.191,A 180.000,B 0.000,C 180.000} C_DIS
LIN {X 72.991,Y 67.274,Z 72.175,A 180.000,B 0.000,C 180.000} C_DIS
LIN {X 73.140,Y 67.223,Z 72.169,A 180.000,B 0.000,C 180.000} C_DIS
LIN {X 73.662,Y 67.047,Z 72.150,A 180.000,B 0.000,C 180.000} C_DIS
LIN {X 74.110,Y 66.896,Z 72.133,A 180.000,B 0.000,C 180.000} C_DIS
LIN {X 74.259,Y 66.846,Z 72.128,A 180.000,B 0.000,C 180.000} C_DIS
LIN {X 74.707,Y 66.695,Z 72.111,A 180.000,B 0.000,C 180.000} C_DIS
LIN {X 74.856,Y 66.644,Z 72.106,A 180.000,B 0.000,C 180.000} C_DIS
LIN {X 75.603,Y 66.392,Z 72.078,A 180.000,B 0.000,C 180.000} C_DIS
LIN {X 75.976,Y 66.267,Z 72.065,A 180.000,B 0.000,C 180.000} C_DIS
LIN {X 76.423,Y 66.116,Z 72.048,A 180.000,B 0.000,C 180.000} C_DIS
LIN {X 77.468,Y 65.763,Z 72.010,A 180.000,B 0.000,C 180.000} C_DIS
LIN {X 77.543,Y 65.737,Z 72.007,A 180.000,B 0.000,C 180.000} C_DIS
LIN {X 77.616,Y 65.710,Z 72.004,A 180.000,B 0.000,C 180.000} C_DIS
LIN {X 77.689,Y 65.680,Z 72.001,A 180.000,B 0.000,C 180.000} C_DIS
LIN {X 77.762,Y 65.648,Z 71.998,A 180.000,B 0.000,C 180.000} C_DIS
LIN {X 77.834,Y 65.614,Z 71.996,A 180.000,B 0.000,C 180.000} C_DIS
LIN {X 77.905,Y 65.577,Z 71.993,A 180.000,B 0.000,C 180.000} C_DIS
LIN {X 77.975,Y 65.539,Z 71.990,A 180.000,B 0.000,C 180.000} C_DIS
LIN {X 78.044,Y 65.499,Z 71.987,A 180.000,B 0.000,C 180.000} C_DIS
LIN {X 78.113,Y 65.455,Z 71.985,A 180.000,B 0.000,C 180.000} C_DIS
LIN {X 78.181,Y 65.410,Z 71.982,A 180.000,B 0.000,C 180.000} C_DIS
LIN {X 78.247,Y 65.363,Z 71.979,A 180.000,B 0.000,C 180.000} C_DIS
LIN {X 78.312,Y 65.314,Z 71.976,A 180.000,B 0.000,C 180.000} C_DIS
LIN {X 78.372,Y 65.267,Z 71.973,A 180.000,B 0.000,C 180.000} C_DIS
LIN {X 78.430,Y 65.217,Z 71.971,A 180.000,B 0.000,C 180.000} C_DIS
LIN {X 78.487,Y 65.166,Z 71.968,A 180.000,B 0.000,C 180.000} C_DIS
LIN {X 78.542,Y 65.114,Z 71.965,A 180.000,B 0.000,C 180.000} C_DIS
LIN {X 78.594,Y 65.063,Z 71.963,A 180.000,B 0.000,C 180.000} C_DIS
LIN {X 78.644,Y 65.011,Z 71.960,A 180.000,B 0.000,C 180.000} C_DIS
LIN {X 78.692,Y 64.957,Z 71.958,A 180.000,B 0.000,C 180.000} C_DIS
LIN {X 78.739,Y 64.902,Z 71.955,A 180.000,B 0.000,C 180.000} C_DIS
LIN {X 78.826,Y 64.793,Z 71.950,A 180.000,B 0.000,C 180.000} C_DIS
LIN {X 78.907,Y 64.680,Z 71.946,A 180.000,B 0.000,C 180.000} C_DIS
LIN {X 78.979,Y 64.568,Z 71.941,A 180.000,B 0.000,C 180.000} C_DIS
LIN {X 79.045,Y 64.453,Z 71.936,A 180.000,B 0.000,C 180.000} C_DIS
LIN {X 79.102,Y 64.341,Z 71.932,A 180.000,B 0.000,C 180.000} C_DIS
LIN {X 79.154,Y 64.227,Z 71.928,A 180.000,B 0.000,C 180.000} C_DIS
LIN {X 79.202,Y 64.109,Z 71.923,A 180.000,B 0.000,C 180.000} C_DIS
LIN {X 79.243,Y 63.988,Z 71.919,A 180.000,B 0.000,C 180.000} C_DIS
LIN {X 79.277,Y 63.873,Z 71.915,A 180.000,B 0.000,C 180.000} C_DIS
LIN {X 79.306,Y 63.757,Z 71.910,A 180.000,B 0.000,C 180.000} C_DIS
LIN {X 79.330,Y 63.635,Z 71.906,A 180.000,B 0.000,C 180.000} C_DIS
LIN {X 79.348,Y 63.512,Z 71.902,A 180.000,B 0.000,C 180.000} C_DIS
LIN {X 79.361,Y 63.392,Z 71.897,A 180.000,B 0.000,C 180.000} C_DIS
LIN {X 79.367,Y 63.271,Z 71.893,A 180.000,B 0.000,C 180.000} C_DIS
LIN {X 79.369,Y 63.158,Z 71.889,A 180.000,B 0.000,C 180.000} C_DIS
LIN {X 79.365,Y 63.046,Z 71.885,A 180.000,B 0.000,C 180.000} C_DIS
LIN {X 79.356,Y 62.932,Z 71.881,A 180.000,B 0.000,C 180.000} C_DIS
LIN {X 79.342,Y 62.819,Z 71.877,A 180.000,B 0.000,C 180.000} C_DIS
LIN {X 79.322,Y 62.699,Z 71.873,A 180.000,B 0.000,C 180.000} C_DIS
LIN {X 79.295,Y 62.580,Z 71.869,A 180.000,B 0.000,C 180.000} C_DIS
LIN {X 79.259,Y 62.442,Z 71.864,A 180.000,B 0.000,C 180.000} C_DIS
LIN {X 79.221,Y 62.305,Z 71.859,A 180.000,B 0.000,C 180.000} C_DIS
LIN {X 79.179,Y 62.152,Z 71.853,A 180.000,B 0.000,C 180.000} C_DIS
LIN {X 79.116,Y 61.924,Z 71.845,A 180.000,B 0.000,C 180.000} C_DIS
LIN {X 79.074,Y 61.772,Z 71.840,A 180.000,B 0.000,C 180.000} C_DIS
LIN {X 79.053,Y 61.696,Z 71.837,A 180.000,B 0.000,C 180.000} C_DIS
LIN {X 79.012,Y 61.544,Z 71.831,A 180.000,B 0.000,C 180.000} C_DIS
LIN {X 78.949,Y 61.316,Z 71.823,A 180.000,B 0.000,C 180.000} C_DIS
LIN {X 78.907,Y 61.164,Z 71.818,A 180.000,B 0.000,C 180.000} C_DIS
LIN {X 78.886,Y 61.088,Z 71.815,A 180.000,B 0.000,C 180.000} C_DIS
LIN {X 78.865,Y 61.012,Z 71.812,A 180.000,B 0.000,C 180.000} C_DIS
LIN {X 78.845,Y 60.935,Z 71.809,A 180.000,B 0.000,C 180.000} C_DIS
LIN {X 78.803,Y 60.783,Z 71.804,A 180.000,B 0.000,C 180.000} C_DIS
LIN {X 78.762,Y 60.631,Z 71.798,A 180.000,B 0.000,C 180.000} C_DIS
LIN {X 78.701,Y 60.402,Z 71.790,A 180.000,B 0.000,C 180.000} C_DIS
LIN {X 78.660,Y 60.250,Z 71.785,A 180.000,B 0.000,C 180.000} C_DIS
LIN {X 78.639,Y 60.174,Z 71.782,A 180.000,B 0.000,C 180.000} C_DIS
LIN {X 78.619,Y 60.097,Z 71.779,A 180.000,B 0.000,C 180.000} C_DIS
LIN {X 78.598,Y 60.021,Z 71.776,A 180.000,B 0.000,C 180.000} C_DIS
LIN {X 78.578,Y 59.945,Z 71.773,A 180.000,B 0.000,C 180.000} C_DIS
LIN {X 78.557,Y 59.869,Z 71.771,A 180.000,B 0.000,C 180.000} C_DIS
LIN {X 78.536,Y 59.793,Z 71.768,A 180.000,B 0.000,C 180.000} C_DIS
LIN {X 78.516,Y 59.717,Z 71.765,A 180.000,B 0.000,C 180.000} C_DIS
LIN {X 78.495,Y 59.640,Z 71.762,A 180.000,B 0.000,C 180.000} C_DIS
LIN {X 78.475,Y 59.564,Z 71.760,A 180.000,B 0.000,C 180.000} C_DIS
LIN {X 78.454,Y 59.488,Z 71.757,A 180.000,B 0.000,C 180.000} C_DIS
LIN {X 78.434,Y 59.412,Z 71.754,A 180.000,B 0.000,C 180.000} C_DIS
LIN {X 78.413,Y 59.336,Z 71.751,A 180.000,B 0.000,C 180.000} C_DIS
LIN {X 78.393,Y 59.259,Z 71.749,A 180.000,B 0.000,C 180.000} C_DIS
LIN {X 78.372,Y 59.183,Z 71.746,A 180.000,B 0.000,C 180.000} C_DIS
LIN {X 78.352,Y 59.107,Z 71.743,A 180.000,B 0.000,C 180.000} C_DIS
LIN {X 78.331,Y 59.031,Z 71.740,A 180.000,B 0.000,C 180.000} C_DIS
LIN {X 78.311,Y 58.955,Z 71.738,A 180.000,B 0.000,C 180.000} C_DIS
LIN {X 78.290,Y 58.879,Z 71.735,A 180.000,B 0.000,C 180.000} C_DIS
LIN {X 78.270,Y 58.802,Z 71.732,A 180.000,B 0.000,C 180.000} C_DIS
LIN {X 78.249,Y 58.726,Z 71.729,A 180.000,B 0.000,C 180.000} C_DIS
LIN {X 78.228,Y 58.650,Z 71.727,A 180.000,B 0.000,C 180.000} C_DIS
LIN {X 78.208,Y 58.574,Z 71.724,A 180.000,B 0.000,C 180.000} C_DIS
LIN {X 78.187,Y 58.498,Z 71.721,A 180.000,B 0.000,C 180.000} C_DIS
LIN {X 78.167,Y 58.421,Z 71.718,A 180.000,B 0.000,C 180.000} C_DIS
LIN {X 78.146,Y 58.345,Z 71.716,A 180.000,B 0.000,C 180.000} C_DIS
LIN {X 78.126,Y 58.269,Z 71.713,A 180.000,B 0.000,C 180.000} C_DIS
LIN {X 78.105,Y 58.193,Z 71.710,A 180.000,B 0.000,C 180.000} C_DIS
LIN {X 78.085,Y 58.117,Z 71.707,A 180.000,B 0.000,C 180.000} C_DIS
LIN {X 78.064,Y 58.041,Z 71.705,A 180.000,B 0.000,C 180.000} C_DIS
LIN {X 78.044,Y 57.964,Z 71.702,A 180.000,B 0.000,C 180.000} C_DIS
LIN {X 78.023,Y 57.888,Z 71.699,A 180.000,B 0.000,C 180.000} C_DIS
LIN {X 78.003,Y 57.812,Z 71.696,A 180.000,B 0.000,C 180.000} C_DIS
LIN {X 77.982,Y 57.736,Z 71.694,A 180.000,B 0.000,C 180.000} C_DIS
LIN {X 77.961,Y 57.660,Z 71.691,A 180.000,B 0.000,C 180.000} C_DIS
LIN {X 77.941,Y 57.583,Z 71.688,A 180.000,B 0.000,C 180.000} C_DIS
LIN {X 77.920,Y 57.507,Z 71.685,A 180.000,B 0.000,C 180.000} C_DIS
LIN {X 77.900,Y 57.431,Z 71.683,A 180.000,B 0.000,C 180.000} C_DIS
LIN {X 77.879,Y 57.355,Z 71.680,A 180.000,B 0.000,C 180.000} C_DIS
LIN {X 77.858,Y 57.279,Z 71.677,A 180.000,B 0.000,C 180.000} C_DIS
LIN {X 77.838,Y 57.203,Z 71.675,A 180.000,B 0.000,C 180.000} C_DIS
LIN {X 77.817,Y 57.127,Z 71.672,A 180.000,B 0.000,C 180.000} C_DIS
LIN {X 77.796,Y 57.050,Z 71.669,A 180.000,B 0.000,C 180.000} C_DIS
LIN {X 77.776,Y 56.974,Z 71.667,A 180.000,B 0.000,C 180.000} C_DIS
LIN {X 77.755,Y 56.898,Z 71.664,A 180.000,B 0.000,C 180.000} C_DIS
LIN {X 77.734,Y 56.822,Z 71.661,A 180.000,B 0.000,C 180.000} C_DIS
LIN {X 77.713,Y 56.746,Z 71.659,A 180.000,B 0.000,C 180.000} C_DIS
LIN {X 77.692,Y 56.670,Z 71.656,A 180.000,B 0.000,C 180.000} C_DIS
LIN {X 77.671,Y 56.594,Z 71.654,A 180.000,B 0.000,C 180.000} C_DIS
LIN {X 77.650,Y 56.518,Z 71.651,A 180.000,B 0.000,C 180.000} C_DIS
LIN {X 77.630,Y 56.442,Z 71.649,A 180.000,B 0.000,C 180.000} C_DIS
LIN {X 77.609,Y 56.366,Z 71.646,A 180.000,B 0.000,C 180.000} C_DIS
LIN {X 77.567,Y 56.214,Z 71.641,A 180.000,B 0.000,C 180.000} C_DIS
LIN {X 77.524,Y 56.062,Z 71.636,A 180.000,B 0.000,C 180.000} C_DIS
LIN {X 77.482,Y 55.910,Z 71.632,A 180.000,B 0.000,C 180.000} C_DIS
LIN {X 77.440,Y 55.758,Z 71.627,A 180.000,B 0.000,C 180.000} C_DIS
LIN {X 77.397,Y 55.606,Z 71.622,A 180.000,B 0.000,C 180.000} C_DIS
LIN {X 77.355,Y 55.454,Z 71.617,A 180.000,B 0.000,C 180.000} C_DIS
LIN {X 77.312,Y 55.302,Z 71.613,A 180.000,B 0.000,C 180.000} C_DIS
LIN {X 77.269,Y 55.151,Z 71.608,A 180.000,B 0.000,C 180.000} C_DIS
LIN {X 77.226,Y 54.999,Z 71.604,A 180.000,B 0.000,C 180.000} C_DIS
LIN {X 77.183,Y 54.847,Z 71.600,A 180.000,B 0.000,C 180.000} C_DIS
LIN {X 77.140,Y 54.695,Z 71.595,A 180.000,B 0.000,C 180.000} C_DIS
LIN {X 77.097,Y 54.544,Z 71.591,A 180.000,B 0.000,C 180.000} C_DIS
LIN {X 77.053,Y 54.392,Z 71.587,A 180.000,B 0.000,C 180.000} C_DIS
LIN {X 77.010,Y 54.241,Z 71.583,A 180.000,B 0.000,C 180.000} C_DIS
LIN {X 76.966,Y 54.089,Z 71.579,A 180.000,B 0.000,C 180.000} C_DIS
LIN {X 76.922,Y 53.938,Z 71.575,A 180.000,B 0.000,C 180.000} C_DIS
LIN {X 76.878,Y 53.786,Z 71.572,A 180.000,B 0.000,C 180.000} C_DIS
LIN {X 76.834,Y 53.635,Z 71.568,A 180.000,B 0.000,C 180.000} C_DIS
LIN {X 76.790,Y 53.484,Z 71.564,A 180.000,B 0.000,C 180.000} C_DIS
LIN {X 76.745,Y 53.333,Z 71.561,A 180.000,B 0.000,C 180.000} C_DIS
LIN {X 76.701,Y 53.181,Z 71.557,A 180.000,B 0.000,C 180.000} C_DIS
LIN {X 76.656,Y 53.030,Z 71.554,A 180.000,B 0.000,C 180.000} C_DIS
LIN {X 76.611,Y 52.879,Z 71.551,A 180.000,B 0.000,C 180.000} C_DIS
LIN {X 76.566,Y 52.728,Z 71.548,A 180.000,B 0.000,C 180.000} C_DIS
LIN {X 76.521,Y 52.577,Z 71.545,A 180.000,B 0.000,C 180.000} C_DIS
LIN {X 76.476,Y 52.426,Z 71.542,A 180.000,B 0.000,C 180.000} C_DIS
LIN {X 76.430,Y 52.275,Z 71.539,A 180.000,B 0.000,C 180.000} C_DIS
LIN {X 76.385,Y 52.125,Z 71.536,A 180.000,B 0.000,C 180.000} C_DIS
LIN {X 76.339,Y 51.974,Z 71.533,A 180.000,B 0.000,C 180.000} C_DIS
LIN {X 76.293,Y 51.823,Z 71.531,A 180.000,B 0.000,C 180.000} C_DIS
LIN {X 76.247,Y 51.672,Z 71.528,A 180.000,B 0.000,C 180.000} C_DIS
LIN {X 76.154,Y 51.371,Z 71.523,A 180.000,B 0.000,C 180.000} C_DIS
LIN {X 76.061,Y 51.070,Z 71.519,A 180.000,B 0.000,C 180.000} C_DIS
LIN {X 75.966,Y 50.770,Z 71.515,A 180.000,B 0.000,C 180.000} C_DIS
LIN {X 75.872,Y 50.469,Z 71.512,A 180.000,B 0.000,C 180.000} C_DIS
LIN {X 75.776,Y 50.169,Z 71.509,A 180.000,B 0.000,C 180.000} C_DIS
LIN {X 75.680,Y 49.869,Z 71.506,A 180.000,B 0.000,C 180.000} C_DIS
LIN {X 75.583,Y 49.569,Z 71.504,A 180.000,B 0.000,C 180.000} C_DIS
LIN {X 75.485,Y 49.270,Z 71.502,A 180.000,B 0.000,C 180.000} C_DIS
LIN {X 75.386,Y 48.971,Z 71.501,A 180.000,B 0.000,C 180.000} C_DIS
LIN {X 75.287,Y 48.672,Z 71.500,A 180.000,B 0.000,C 180.000} C_DIS
LIN {X 75.185,Y 48.369,Z 71.500,A 180.000,B 0.000,C 180.000} C_DIS
; Cutting Move Starts
LIN {X 73.524,Y 43.444,Z 71.500,A 180.000,B 0.000,C 180.000} C_DIS
LIN {X 73.478,Y 43.310,Z 71.500,A 180.000,B 0.000,C 180.000} C_DIS
LIN {X 73.461,Y 43.266,Z 71.500,A 180.000,B 0.000,C 180.000} C_DIS
LIN {X 73.385,Y 43.087,Z 71.500,A 180.000,B 0.000,C 180.000} C_DIS
LIN {X 73.299,Y 42.921,Z 71.500,A 180.000,B 0.000,C 180.000} C_DIS
LIN {X 73.291,Y 42.908,Z 71.500,A 180.000,B 0.000,C 180.000} C_DIS
LIN {X 73.178,Y 42.729,Z 71.500,A 180.000,B 0.000,C 180.000} C_DIS
LIN {X 73.120,Y 42.650,Z 71.500,A 180.000,B 0.000,C 180.000} C_DIS
LIN {X 73.041,Y 42.550,Z 71.500,A 180.000,B 0.000,C 180.000} C_DIS
LIN {X 72.941,Y 42.439,Z 71.500,A 180.000,B 0.000,C 180.000} C_DIS
LIN {X 72.876,Y 42.372,Z 71.500,A 180.000,B 0.000,C 180.000} C_DIS
LIN {X 72.763,Y 42.268,Z 71.500,A 180.000,B 0.000,C 180.000} C_DIS
LIN {X 72.672,Y 42.193,Z 71.500,A 180.000,B 0.000,C 180.000} C_DIS
LIN {X 72.584,Y 42.126,Z 71.500,A 180.000,B 0.000,C 180.000} C_DIS
LIN {X 72.413,Y 42.014,Z 71.500,A 180.000,B 0.000,C 180.000} C_DIS
LIN {X 72.405,Y 42.009,Z 71.500,A 180.000,B 0.000,C 180.000} C_DIS
LIN {X 72.226,Y 41.912,Z 71.500,A 180.000,B 0.000,C 180.000} C_DIS
LIN {X 72.053,Y 41.835,Z 71.500,A 180.000,B 0.000,C 180.000} C_DIS
LIN {X 72.048,Y 41.833,Z 71.500,A 180.000,B 0.000,C 180.000} C_DIS
LIN {X 71.869,Y 41.770,Z 71.500,A 180.000,B 0.000,C 180.000} C_DIS
LIN {X 71.690,Y 41.722,Z 71.500,A 180.000,B 0.000,C 180.000} C_DIS
LIN {X 71.511,Y 41.687,Z 71.500,A 180.000,B 0.000,C 180.000} C_DIS
LIN {X 71.422,Y 41.675,Z 71.500,A 180.000,B 0.000,C 180.000} C_DIS
LIN {X 71.332,Y 41.666,Z 71.500,A 180.000,B 0.000,C 180.000} C_DIS
LIN {X 71.243,Y 41.660,Z 71.500,A 180.000,B 0.000,C 180.000} C_DIS
LIN {X 71.154,Y 41.657,Z 71.500,A 180.000,B 0.000,C 180.000} C_DIS
LIN {X 71.064,Y 41.658,Z 71.500,A 180.000,B 0.000,C 180.000} C_DIS
LIN {X 70.975,Y 41.662,Z 71.500,A 180.000,B 0.000,C 180.000} C_DIS
LIN {X 70.886,Y 41.669,Z 71.500,A 180.000,B 0.000,C 180.000} C_DIS
LIN {X 70.796,Y 41.679,Z 71.500,A 180.000,B 0.000,C 180.000} C_DIS
LIN {X 70.707,Y 41.692,Z 71.500,A 180.000,B 0.000,C 180.000} C_DIS
LIN {X 70.617,Y 41.709,Z 71.500,A 180.000,B 0.000,C 180.000} C_DIS
LIN {X 70.528,Y 41.729,Z 71.500,A 180.000,B 0.000,C 180.000} C_DIS
LIN {X 70.439,Y 41.753,Z 71.500,A 180.000,B 0.000,C 180.000} C_DIS
LIN {X 70.349,Y 41.781,Z 71.500,A 180.000,B 0.000,C 180.000} C_DIS
LIN {X 70.260,Y 41.811,Z 71.500,A 180.000,B 0.000,C 180.000} C_DIS
LIN {X 45.590,Y 50.133,Z 71.500,A 180.000,B 0.000,C 180.000} C_DIS
LIN {X 45.411,Y 50.194,Z 71.500,A 180.000,B 0.000,C 180.000} C_DIS
LIN {X 45.296,Y 50.238,Z 71.500,A 180.000,B 0.000,C 180.000} C_DIS
LIN {X 45.232,Y 50.265,Z 71.500,A 180.000,B 0.000,C 180.000} C_DIS
LIN {X 45.053,Y 50.353,Z 71.500,A 180.000,B 0.000,C 180.000} C_DIS
LIN {X 44.944,Y 50.416,Z 71.500,A 180.000,B 0.000,C 180.000} C_DIS
LIN {X 44.874,Y 50.461,Z 71.500,A 180.000,B 0.000,C 180.000} C_DIS
LIN {X 44.785,Y 50.522,Z 71.500,A 180.000,B 0.000,C 180.000} C_DIS
LIN {X 44.696,Y 50.590,Z 71.500,A 180.000,B 0.000,C 180.000} C_DIS
LIN {X 44.689,Y 50.595,Z 71.500,A 180.000,B 0.000,C 180.000} C_DIS
LIN {X 44.603,Y 50.667,Z 71.500,A 180.000,B 0.000,C 180.000} C_DIS
LIN {X 44.517,Y 50.746,Z 71.500,A 180.000,B 0.000,C 180.000} C_DIS
LIN {X 44.488,Y 50.774,Z 71.500,A 180.000,B 0.000,C 180.000} C_DIS
LIN {X 44.410,Y 50.855,Z 71.500,A 180.000,B 0.000,C 180.000} C_DIS
LIN {X 44.338,Y 50.936,Z 71.500,A 180.000,B 0.000,C 180.000} C_DIS
LIN {X 44.325,Y 50.953,Z 71.500,A 180.000,B 0.000,C 180.000} C_DIS
LIN {X 44.254,Y 51.042,Z 71.500,A 180.000,B 0.000,C 180.000} C_DIS
LIN {X 44.189,Y 51.131,Z 71.500,A 180.000,B 0.000,C 180.000} C_DIS
LIN {X 44.159,Y 51.176,Z 71.500,A 180.000,B 0.000,C 180.000} C_DIS
LIN {X 44.077,Y 51.310,Z 71.500,A 180.000,B 0.000,C 180.000} C_DIS
LIN {X 43.984,Y 51.489,Z 71.500,A 180.000,B 0.000,C 180.000} C_DIS
LIN {X 43.981,Y 51.497,Z 71.500,A 180.000,B 0.000,C 180.000} C_DIS
LIN {X 43.909,Y 51.668,Z 71.500,A 180.000,B 0.000,C 180.000} C_DIS
LIN {X 43.849,Y 51.847,Z 71.500,A 180.000,B 0.000,C 180.000} C_DIS
LIN {X 43.804,Y 52.025,Z 71.500,A 180.000,B 0.000,C 180.000} C_DIS
LIN {X 43.802,Y 52.035,Z 71.500,A 180.000,B 0.000,C 180.000} C_DIS
LIN {X 43.772,Y 52.204,Z 71.500,A 180.000,B 0.000,C 180.000} C_DIS
LIN {X 43.754,Y 52.383,Z 71.500,A 180.000,B 0.000,C 180.000} C_DIS
LIN {X 43.748,Y 52.562,Z 71.500,A 180.000,B 0.000,C 180.000} C_DIS
LIN {X 43.756,Y 52.740,Z 71.500,A 180.000,B 0.000,C 180.000} C_DIS
LIN {X 43.776,Y 52.919,Z 71.500,A 180.000,B 0.000,C 180.000} C_DIS
LIN {X 43.802,Y 53.064,Z 71.500,A 180.000,B 0.000,C 180.000} C_DIS
LIN {X 43.809,Y 53.098,Z 71.500,A 180.000,B 0.000,C 180.000} C_DIS
LIN {X 43.856,Y 53.277,Z 71.500,A 180.000,B 0.000,C 180.000} C_DIS
LIN {X 43.916,Y 53.455,Z 71.500,A 180.000,B 0.000,C 180.000} C_DIS
LIN {X 50.248,Y 72.226,Z 71.500,A 180.000,B 0.000,C 180.000} C_DIS
LIN {X 50.311,Y 72.405,Z 71.500,A 180.000,B 0.000,C 180.000} C_DIS
LIN {X 50.388,Y 72.584,Z 71.500,A 180.000,B 0.000,C 180.000} C_DIS
LIN {X 50.416,Y 72.640,Z 71.500,A 180.000,B 0.000,C 180.000} C_DIS
LIN {X 50.484,Y 72.763,Z 71.500,A 180.000,B 0.000,C 180.000} C_DIS
LIN {X 50.595,Y 72.936,Z 71.500,A 180.000,B 0.000,C 180.000} C_DIS
LIN {X 50.599,Y 72.941,Z 71.500,A 180.000,B 0.000,C 180.000} C_DIS
LIN {X 50.665,Y 73.031,Z 71.500,A 180.000,B 0.000,C 180.000} C_DIS
LIN {X 50.737,Y 73.120,Z 71.500,A 180.000,B 0.000,C 180.000} C_DIS
LIN {X 50.774,Y 73.162,Z 71.500,A 180.000,B 0.000,C 180.000} C_DIS
LIN {X 50.905,Y 73.299,Z 71.500,A 180.000,B 0.000,C 180.000} C_DIS
LIN {X 50.953,Y 73.343,Z 71.500,A 180.000,B 0.000,C 180.000} C_DIS
LIN {X 51.112,Y 73.478,Z 71.500,A 180.000,B 0.000,C 180.000} C_DIS
LIN {X 51.131,Y 73.493,Z 71.500,A 180.000,B 0.000,C 180.000} C_DIS
LIN {X 51.310,Y 73.616,Z 71.500,A 180.000,B 0.000,C 180.000} C_DIS
LIN {X 51.376,Y 73.656,Z 71.500,A 180.000,B 0.000,C 180.000} C_DIS
LIN {X 51.489,Y 73.719,Z 71.500,A 180.000,B 0.000,C 180.000} C_DIS
LIN {X 51.668,Y 73.803,Z 71.500,A 180.000,B 0.000,C 180.000} C_DIS
LIN {X 51.749,Y 73.835,Z 71.500,A 180.000,B 0.000,C 180.000} C_DIS
LIN {X 51.847,Y 73.870,Z 71.500,A 180.000,B 0.000,C 180.000} C_DIS
LIN {X 52.025,Y 73.923,Z 71.500,A 180.000,B 0.000,C 180.000} C_DIS
LIN {X 52.204,Y 73.961,Z 71.500,A 180.000,B 0.000,C 180.000} C_DIS
LIN {X 52.383,Y 73.987,Z 71.500,A 180.000,B 0.000,C 180.000} C_DIS
LIN {X 52.562,Y 73.999,Z 71.500,A 180.000,B 0.000,C 180.000} C_DIS
LIN {X 52.740,Y 73.998,Z 71.500,A 180.000,B 0.000,C 180.000} C_DIS
LIN {X 52.919,Y 73.985,Z 71.500,A 180.000,B 0.000,C 180.000} C_DIS
LIN {X 53.098,Y 73.958,Z 71.500,A 180.000,B 0.000,C 180.000} C_DIS
LIN {X 53.277,Y 73.918,Z 71.500,A 180.000,B 0.000,C 180.000} C_DIS
LIN {X 53.455,Y 73.864,Z 71.500,A 180.000,B 0.000,C 180.000} C_DIS
LIN {X 57.977,Y 72.338,Z 71.500,A 180.000,B 0.000,C 180.000} C_DIS
LIN {X 78.304,Y 65.481,Z 71.500,A 180.000,B 0.000,C 180.000} C_DIS
LIN {X 78.371,Y 65.458,Z 71.500,A 180.000,B 0.000,C 180.000} C_DIS
LIN {X 78.437,Y 65.433,Z 71.500,A 180.000,B 0.000,C 180.000} C_DIS
LIN {X 78.483,Y 65.414,Z 71.500,A 180.000,B 0.000,C 180.000} C_DIS
LIN {X 78.573,Y 65.375,Z 71.500,A 180.000,B 0.000,C 180.000} C_DIS
LIN {X 78.662,Y 65.331,Z 71.500,A 180.000,B 0.000,C 180.000} C_DIS
LIN {X 78.731,Y 65.294,Z 71.500,A 180.000,B 0.000,C 180.000} C_DIS
LIN {X 78.800,Y 65.254,Z 71.500,A 180.000,B 0.000,C 180.000} C_DIS
LIN {X 78.841,Y 65.229,Z 71.500,A 180.000,B 0.000,C 180.000} C_DIS
LIN {X 78.930,Y 65.171,Z 71.500,A 180.000,B 0.000,C 180.000} C_DIS
LIN {X 79.020,Y 65.107,Z 71.500,A 180.000,B 0.000,C 180.000} C_DIS
LIN {X 79.061,Y 65.075,Z 71.500,A 180.000,B 0.000,C 180.000} C_DIS
LIN {X 79.129,Y 65.020,Z 71.500,A 180.000,B 0.000,C 180.000} C_DIS
LIN {X 79.198,Y 64.959,Z 71.500,A 180.000,B 0.000,C 180.000} C_DIS
LIN {X 79.265,Y 64.897,Z 71.500,A 180.000,B 0.000,C 180.000} C_DIS
LIN {X 79.377,Y 64.780,Z 71.500,A 180.000,B 0.000,C 180.000} C_DIS
LIN {X 79.431,Y 64.718,Z 71.500,A 180.000,B 0.000,C 180.000} C_DIS
LIN {X 79.556,Y 64.557,Z 71.500,A 180.000,B 0.000,C 180.000} C_DIS
LIN {X 79.568,Y 64.539,Z 71.500,A 180.000,B 0.000,C 180.000} C_DIS
LIN {X 79.682,Y 64.360,Z 71.500,A 180.000,B 0.000,C 180.000} C_DIS
LIN {X 79.735,Y 64.265,Z 71.500,A 180.000,B 0.000,C 180.000} C_DIS
LIN {X 79.776,Y 64.182,Z 71.500,A 180.000,B 0.000,C 180.000} C_DIS
LIN {X 79.853,Y 64.003,Z 71.500,A 180.000,B 0.000,C 180.000} C_DIS
LIN {X 79.913,Y 63.825,Z 71.500,A 180.000,B 0.000,C 180.000} C_DIS
LIN {X 79.914,Y 63.824,Z 71.500,A 180.000,B 0.000,C 180.000} C_DIS
LIN {X 79.960,Y 63.645,Z 71.500,A 180.000,B 0.000,C 180.000} C_DIS
LIN {X 79.993,Y 63.467,Z 71.500,A 180.000,B 0.000,C 180.000} C_DIS
LIN {X 80.012,Y 63.288,Z 71.500,A 180.000,B 0.000,C 180.000} C_DIS
LIN {X 80.019,Y 63.109,Z 71.500,A 180.000,B 0.000,C 180.000} C_DIS
LIN {X 80.012,Y 62.930,Z 71.500,A 180.000,B 0.000,C 180.000} C_DIS
LIN {X 79.993,Y 62.751,Z 71.500,A 180.000,B 0.000,C 180.000} C_DIS
LIN {X 79.961,Y 62.573,Z 71.500,A 180.000,B 0.000,C 180.000} C_DIS
LIN {X 79.915,Y 62.394,Z 71.500,A 180.000,B 0.000,C 180.000} C_DIS
LIN {X 79.913,Y 62.390,Z 71.500,A 180.000,B 0.000,C 180.000} C_DIS
LIN {X 79.856,Y 62.215,Z 71.500,A 180.000,B 0.000,C 180.000} C_DIS
LIN {X 75.185,Y 48.369,Z 71.500,A 180.000,B 0.000,C 180.000} C_DIS
; Lead Out Move Starts
LIN {X 75.330,Y 47.832,Z 71.500,A 180.000,B 0.000,C 180.000} C_DIS
LIN {X 75.881,Y 47.761,Z 71.500,A 180.000,B 0.000,C 180.000} C_DIS
; Rapid Move Starts
LIN {X 75.881,Y 47.761,Z 95.000,A 180.000,B 0.000,C 180.000} C_DIS
LIN {X 81.999,Y 45.697,Z 95.000,A 180.000,B 0.000,C 180.000} C_DIS
LIN {X 81.999,Y 45.697,Z 75.399,A 180.000,B 0.000,C 180.000} C_DIS
; Plunge Move Starts
$VEL.CP=0.01
LIN {X 81.999,Y 45.697,Z 74.625,A 180.000,B 0.000,C 180.000} C_DIS
; Lead In Move Starts
LIN {X 81.999,Y 45.697,Z 73.500,A 180.000,B 0.000,C 180.000} C_DIS
LIN {X 82.481,Y 45.420,Z 73.500,A 180.000,B 0.000,C 180.000} C_DIS
LIN {X 82.921,Y 45.759,Z 73.500,A 180.000,B 0.000,C 180.000} C_DIS
; Cutting Move Starts
$VEL.CP=0.02
LIN {X 87.601,Y 59.630,Z 73.500,A 180.000,B 0.000,C 180.000} C_DIS
LIN {X 87.628,Y 59.712,Z 73.500,A 180.000,B 0.000,C 180.000} C_DIS
LIN {X 87.698,Y 59.891,Z 73.500,A 180.000,B 0.000,C 180.000} C_DIS
LIN {X 87.779,Y 60.062,Z 73.500,A 180.000,B 0.000,C 180.000} C_DIS
LIN {X 87.783,Y 60.070,Z 73.500,A 180.000,B 0.000,C 180.000} C_DIS
LIN {X 87.888,Y 60.249,Z 73.500,A 180.000,B 0.000,C 180.000} C_DIS
LIN {X 87.958,Y 60.352,Z 73.500,A 180.000,B 0.000,C 180.000} C_DIS
LIN {X 88.014,Y 60.427,Z 73.500,A 180.000,B 0.000,C 180.000} C_DIS
LIN {X 88.137,Y 60.575,Z 73.500,A 180.000,B 0.000,C 180.000} C_DIS
LIN {X 88.166,Y 60.606,Z 73.500,A 180.000,B 0.000,C 180.000} C_DIS
LIN {X 88.316,Y 60.754,Z 73.500,A 180.000,B 0.000,C 180.000} C_DIS
LIN {X 88.351,Y 60.785,Z 73.500,A 180.000,B 0.000,C 180.000} C_DIS
LIN {X 88.494,Y 60.901,Z 73.500,A 180.000,B 0.000,C 180.000} C_DIS
LIN {X 88.582,Y 60.964,Z 73.500,A 180.000,B 0.000,C 180.000} C_DIS
LIN {X 88.673,Y 61.023,Z 73.500,A 180.000,B 0.000,C 180.000} C_DIS
LIN {X 88.852,Y 61.124,Z 73.500,A 180.000,B 0.000,C 180.000} C_DIS
LIN {X 88.889,Y 61.143,Z 73.500,A 180.000,B 0.000,C 180.000} C_DIS
LIN {X 89.031,Y 61.207,Z 73.500,A 180.000,B 0.000,C 180.000} C_DIS
LIN {X 89.209,Y 61.274,Z 73.500,A 180.000,B 0.000,C 180.000} C_DIS
LIN {X 89.372,Y 61.321,Z 73.500,A 180.000,B 0.000,C 180.000} C_DIS
LIN {X 89.388,Y 61.325,Z 73.500,A 180.000,B 0.000,C 180.000} C_DIS
LIN {X 89.567,Y 61.363,Z 73.500,A 180.000,B 0.000,C 180.000} C_DIS
LIN {X 89.656,Y 61.377,Z 73.500,A 180.000,B 0.000,C 180.000} C_DIS
LIN {X 89.746,Y 61.387,Z 73.500,A 180.000,B 0.000,C 180.000} C_DIS
LIN {X 89.835,Y 61.395,Z 73.500,A 180.000,B 0.000,C 180.000} C_DIS
LIN {X 89.925,Y 61.399,Z 73.500,A 180.000,B 0.000,C 180.000} C_DIS
LIN {X 90.014,Y 61.399,Z 73.500,A 180.000,B 0.000,C 180.000} C_DIS
LIN {X 90.103,Y 61.397,Z 73.500,A 180.000,B 0.000,C 180.000} C_DIS
LIN {X 90.193,Y 61.392,Z 73.500,A 180.000,B 0.000,C 180.000} C_DIS
LIN {X 90.282,Y 61.383,Z 73.500,A 180.000,B 0.000,C 180.000} C_DIS
LIN {X 90.371,Y 61.371,Z 73.500,A 180.000,B 0.000,C 180.000} C_DIS
LIN {X 90.461,Y 61.355,Z 73.500,A 180.000,B 0.000,C 180.000} C_DIS
LIN {X 90.537,Y 61.340,Z 73.500,A 180.000,B 0.000,C 180.000} C_DIS
LIN {X 90.613,Y 61.321,Z 73.500,A 180.000,B 0.000,C 180.000} C_DIS
LIN {X 90.640,Y 61.314,Z 73.500,A 180.000,B 0.000,C 180.000} C_DIS
LIN {X 90.729,Y 61.289,Z 73.500,A 180.000,B 0.000,C 180.000} C_DIS
LIN {X 90.818,Y 61.259,Z 73.500,A 180.000,B 0.000,C 180.000} C_DIS
LIN {X 93.589,Y 60.325,Z 73.500,A 180.000,B 0.000,C 180.000} C_DIS
LIN {X 93.634,Y 60.309,Z 73.500,A 180.000,B 0.000,C 180.000} C_DIS
LIN {X 93.679,Y 60.293,Z 73.500,A 180.000,B 0.000,C 180.000} C_DIS
LIN {X 93.733,Y 60.271,Z 73.500,A 180.000,B 0.000,C 180.000} C_DIS
LIN {X 93.787,Y 60.249,Z 73.500,A 180.000,B 0.000,C 180.000} C_DIS
LIN {X 93.857,Y 60.217,Z 73.500,A 180.000,B 0.000,C 180.000} C_DIS
LIN {X 93.902,Y 60.196,Z 73.500,A 180.000,B 0.000,C 180.000} C_DIS
LIN {X 93.947,Y 60.173,Z 73.500,A 180.000,B 0.000,C 180.000} C_DIS
LIN {X 93.992,Y 60.149,Z 73.500,A 180.000,B 0.000,C 180.000} C_DIS
LIN {X 94.036,Y 60.124,Z 73.500,A 180.000,B 0.000,C 180.000} C_DIS
LIN {X 94.127,Y 60.070,Z 73.500,A 180.000,B 0.000,C 180.000} C_DIS
LIN {X 94.215,Y 60.012,Z 73.500,A 180.000,B 0.000,C 180.000} C_DIS
LIN {X 94.295,Y 59.954,Z 73.500,A 180.000,B 0.000,C 180.000} C_DIS
LIN {X 94.375,Y 59.891,Z 73.500,A 180.000,B 0.000,C 180.000} C_DIS
LIN {X 94.394,Y 59.876,Z 73.500,A 180.000,B 0.000,C 180.000} C_DIS
LIN {X 94.483,Y 59.798,Z 73.500,A 180.000,B 0.000,C 180.000} C_DIS
LIN {X 94.572,Y 59.712,Z 73.500,A 180.000,B 0.000,C 180.000} C_DIS
LIN {X 94.573,Y 59.712,Z 73.500,A 180.000,B 0.000,C 180.000} C_DIS
LIN {X 94.656,Y 59.623,Z 73.500,A 180.000,B 0.000,C 180.000} C_DIS
LIN {X 94.733,Y 59.534,Z 73.500,A 180.000,B 0.000,C 180.000} C_DIS
LIN {X 94.751,Y 59.510,Z 73.500,A 180.000,B 0.000,C 180.000} C_DIS
LIN {X 94.865,Y 59.355,Z 73.500,A 180.000,B 0.000,C 180.000} C_DIS
LIN {X 94.930,Y 59.254,Z 73.500,A 180.000,B 0.000,C 180.000} C_DIS
LIN {X 94.976,Y 59.176,Z 73.500,A 180.000,B 0.000,C 180.000} C_DIS
LIN {X 95.067,Y 58.997,Z 73.500,A 180.000,B 0.000,C 180.000} C_DIS
LIN {X 95.109,Y 58.900,Z 73.500,A 180.000,B 0.000,C 180.000} C_DIS
LIN {X 95.141,Y 58.819,Z 73.500,A 180.000,B 0.000,C 180.000} C_DIS
LIN {X 95.199,Y 58.640,Z 73.500,A 180.000,B 0.000,C 180.000} C_DIS
LIN {X 95.243,Y 58.461,Z 73.500,A 180.000,B 0.000,C 180.000} C_DIS
LIN {X 95.273,Y 58.282,Z 73.500,A 180.000,B 0.000,C 180.000} C_DIS
LIN {X 95.288,Y 58.142,Z 73.500,A 180.000,B 0.000,C 180.000} C_DIS
LIN {X 95.290,Y 58.103,Z 73.500,A 180.000,B 0.000,C 180.000} C_DIS
LIN {X 95.294,Y 57.925,Z 73.500,A 180.000,B 0.000,C 180.000} C_DIS
LIN {X 95.288,Y 57.767,Z 73.500,A 180.000,B 0.000,C 180.000} C_DIS
LIN {X 95.286,Y 57.746,Z 73.500,A 180.000,B 0.000,C 180.000} C_DIS
LIN {X 95.264,Y 57.567,Z 73.500,A 180.000,B 0.000,C 180.000} C_DIS
LIN {X 95.230,Y 57.388,Z 73.500,A 180.000,B 0.000,C 180.000} C_DIS
LIN {X 95.181,Y 57.210,Z 73.500,A 180.000,B 0.000,C 180.000} C_DIS
LIN {X 95.122,Y 57.031,Z 73.500,A 180.000,B 0.000,C 180.000} C_DIS
LIN {X 88.789,Y 38.260,Z 73.500,A 180.000,B 0.000,C 180.000} C_DIS
LIN {X 88.725,Y 38.081,Z 73.500,A 180.000,B 0.000,C 180.000} C_DIS
LIN {X 88.673,Y 37.959,Z 73.500,A 180.000,B 0.000,C 180.000} C_DIS
LIN {X 88.646,Y 37.902,Z 73.500,A 180.000,B 0.000,C 180.000} C_DIS
LIN {X 88.549,Y 37.724,Z 73.500,A 180.000,B 0.000,C 180.000} C_DIS
LIN {X 88.494,Y 37.636,Z 73.500,A 180.000,B 0.000,C 180.000} C_DIS
LIN {X 88.432,Y 37.545,Z 73.500,A 180.000,B 0.000,C 180.000} C_DIS
LIN {X 88.316,Y 37.395,Z 73.500,A 180.000,B 0.000,C 180.000} C_DIS
LIN {X 88.291,Y 37.366,Z 73.500,A 180.000,B 0.000,C 180.000} C_DIS
LIN {X 88.137,Y 37.204,Z 73.500,A 180.000,B 0.000,C 180.000} C_DIS
LIN {X 88.120,Y 37.187,Z 73.500,A 180.000,B 0.000,C 180.000} C_DIS
LIN {X 87.958,Y 37.047,Z 73.500,A 180.000,B 0.000,C 180.000} C_DIS
LIN {X 87.908,Y 37.009,Z 73.500,A 180.000,B 0.000,C 180.000} C_DIS
LIN {X 87.779,Y 36.917,Z 73.500,A 180.000,B 0.000,C 180.000} C_DIS
LIN {X 87.636,Y 36.830,Z 73.500,A 180.000,B 0.000,C 180.000} C_DIS
LIN {X 87.601,Y 36.810,Z 73.500,A 180.000,B 0.000,C 180.000} C_DIS
LIN {X 87.422,Y 36.721,Z 73.500,A 180.000,B 0.000,C 180.000} C_DIS
LIN {X 87.248,Y 36.651,Z 73.500,A 180.000,B 0.000,C 180.000} C_DIS
LIN {X 87.243,Y 36.649,Z 73.500,A 180.000,B 0.000,C 180.000} C_DIS
LIN {X 87.064,Y 36.593,Z 73.500,A 180.000,B 0.000,C 180.000} C_DIS
LIN {X 86.885,Y 36.551,Z 73.500,A 180.000,B 0.000,C 180.000} C_DIS
LIN {X 86.707,Y 36.522,Z 73.500,A 180.000,B 0.000,C 180.000} C_DIS
LIN {X 86.617,Y 36.513,Z 73.500,A 180.000,B 0.000,C 180.000} C_DIS
LIN {X 86.528,Y 36.507,Z 73.500,A 180.000,B 0.000,C 180.000} C_DIS
LIN {X 86.438,Y 36.504,Z 73.500,A 180.000,B 0.000,C 180.000} C_DIS
LIN {X 86.349,Y 36.504,Z 73.500,A 180.000,B 0.000,C 180.000} C_DIS
LIN {X 86.260,Y 36.508,Z 73.500,A 180.000,B 0.000,C 180.000} C_DIS
LIN {X 86.170,Y 36.514,Z 73.500,A 180.000,B 0.000,C 180.000} C_DIS
LIN {X 86.081,Y 36.524,Z 73.500,A 180.000,B 0.000,C 180.000} C_DIS
LIN {X 85.992,Y 36.537,Z 73.500,A 180.000,B 0.000,C 180.000} C_DIS
LIN {X 85.902,Y 36.554,Z 73.500,A 180.000,B 0.000,C 180.000} C_DIS
LIN {X 85.813,Y 36.574,Z 73.500,A 180.000,B 0.000,C 180.000} C_DIS
LIN {X 85.768,Y 36.585,Z 73.500,A 180.000,B 0.000,C 180.000} C_DIS
LIN {X 85.723,Y 36.597,Z 73.500,A 180.000,B 0.000,C 180.000} C_DIS
LIN {X 85.679,Y 36.610,Z 73.500,A 180.000,B 0.000,C 180.000} C_DIS
LIN {X 85.634,Y 36.624,Z 73.500,A 180.000,B 0.000,C 180.000} C_DIS
LIN {X 85.554,Y 36.651,Z 73.500,A 180.000,B 0.000,C 180.000} C_DIS
LIN {X 82.905,Y 37.545,Z 73.500,A 180.000,B 0.000,C 180.000} C_DIS
LIN {X 82.774,Y 37.589,Z 73.500,A 180.000,B 0.000,C 180.000} C_DIS
LIN {X 82.684,Y 37.622,Z 73.500,A 180.000,B 0.000,C 180.000} C_DIS
LIN {X 82.595,Y 37.660,Z 73.500,A 180.000,B 0.000,C 180.000} C_DIS
LIN {X 82.527,Y 37.690,Z 73.500,A 180.000,B 0.000,C 180.000} C_DIS
LIN {X 82.460,Y 37.724,Z 73.500,A 180.000,B 0.000,C 180.000} C_DIS
LIN {X 82.416,Y 37.747,Z 73.500,A 180.000,B 0.000,C 180.000} C_DIS
LIN {X 82.327,Y 37.797,Z 73.500,A 180.000,B 0.000,C 180.000} C_DIS
LIN {X 82.237,Y 37.853,Z 73.500,A 180.000,B 0.000,C 180.000} C_DIS
LIN {X 82.164,Y 37.902,Z 73.500,A 180.000,B 0.000,C 180.000} C_DIS
LIN {X 82.059,Y 37.980,Z 73.500,A 180.000,B 0.000,C 180.000} C_DIS
LIN {X 81.938,Y 38.081,Z 73.500,A 180.000,B 0.000,C 180.000} C_DIS
LIN {X 81.880,Y 38.134,Z 73.500,A 180.000,B 0.000,C 180.000} C_DIS
LIN {X 81.756,Y 38.260,Z 73.500,A 180.000,B 0.000,C 180.000} C_DIS
LIN {X 81.701,Y 38.322,Z 73.500,A 180.000,B 0.000,C 180.000} C_DIS
LIN {X 81.607,Y 38.439,Z 73.500,A 180.000,B 0.000,C 180.000} C_DIS
LIN {X 81.522,Y 38.558,Z 73.500,A 180.000,B 0.000,C 180.000} C_DIS
LIN {X 81.484,Y 38.618,Z 73.500,A 180.000,B 0.000,C 180.000} C_DIS
LIN {X 81.381,Y 38.796,Z 73.500,A 180.000,B 0.000,C 180.000} C_DIS
LIN {X 81.344,Y 38.872,Z 73.500,A 180.000,B 0.000,C 180.000} C_DIS
LIN {X 81.297,Y 38.975,Z 73.500,A 180.000,B 0.000,C 180.000} C_DIS
LIN {X 81.229,Y 39.154,Z 73.500,A 180.000,B 0.000,C 180.000} C_DIS
LIN {X 81.177,Y 39.333,Z 73.500,A 180.000,B 0.000,C 180.000} C_DIS
LIN {X 81.165,Y 39.382,Z 73.500,A 180.000,B 0.000,C 180.000} C_DIS
LIN {X 81.138,Y 39.511,Z 73.500,A 180.000,B 0.000,C 180.000} C_DIS
LIN {X 81.113,Y 39.690,Z 73.500,A 180.000,B 0.000,C 180.000} C_DIS
LIN {X 81.101,Y 39.869,Z 73.500,A 180.000,B 0.000,C 180.000} C_DIS
LIN {X 81.102,Y 40.048,Z 73.500,A 180.000,B 0.000,C 180.000} C_DIS
LIN {X 81.115,Y 40.226,Z 73.500,A 180.000,B 0.000,C 180.000} C_DIS
LIN {X 81.142,Y 40.405,Z 73.500,A 180.000,B 0.000,C 180.000} C_DIS
LIN {X 81.165,Y 40.516,Z 73.500,A 180.000,B 0.000,C 180.000} C_DIS
LIN {X 81.182,Y 40.584,Z 73.500,A 180.000,B 0.000,C 180.000} C_DIS
LIN {X 81.236,Y 40.763,Z 73.500,A 180.000,B 0.000,C 180.000} C_DIS
LIN {X 82.921,Y 45.759,Z 73.500,A 180.000,B 0.000,C 180.000} C_DIS
; Link Move Starts
LIN {X 83.022,Y 46.057,Z 73.500,A 180.000,B 0.000,C 180.000} C_DIS
LIN {X 83.121,Y 46.356,Z 73.499,A 180.000,B 0.000,C 180.000} C_DIS
LIN {X 83.221,Y 46.655,Z 73.498,A 180.000,B 0.000,C 180.000} C_DIS
LIN {X 83.319,Y 46.954,Z 73.496,A 180.000,B 0.000,C 180.000} C_DIS
LIN {X 83.418,Y 47.253,Z 73.494,A 180.000,B 0.000,C 180.000} C_DIS
LIN {X 83.515,Y 47.553,Z 73.491,A 180.000,B 0.000,C 180.000} C_DIS
LIN {X 83.613,Y 47.852,Z 73.488,A 180.000,B 0.000,C 180.000} C_DIS
LIN {X 83.709,Y 48.152,Z 73.485,A 180.000,B 0.000,C 180.000} C_DIS
LIN {X 83.806,Y 48.452,Z 73.481,A 180.000,B 0.000,C 180.000} C_DIS
LIN {X 83.901,Y 48.752,Z 73.477,A 180.000,B 0.000,C 180.000} C_DIS
LIN {X 83.997,Y 49.053,Z 73.472,A 180.000,B 0.000,C 180.000} C_DIS
LIN {X 84.044,Y 49.203,Z 73.469,A 180.000,B 0.000,C 180.000} C_DIS
LIN {X 84.092,Y 49.353,Z 73.467,A 180.000,B 0.000,C 180.000} C_DIS
LIN {X 84.139,Y 49.503,Z 73.464,A 180.000,B 0.000,C 180.000} C_DIS
LIN {X 84.186,Y 49.654,Z 73.461,A 180.000,B 0.000,C 180.000} C_DIS
LIN {X 84.233,Y 49.804,Z 73.459,A 180.000,B 0.000,C 180.000} C_DIS
LIN {X 84.280,Y 49.954,Z 73.456,A 180.000,B 0.000,C 180.000} C_DIS
LIN {X 84.327,Y 50.105,Z 73.452,A 180.000,B 0.000,C 180.000} C_DIS
LIN {X 84.374,Y 50.255,Z 73.449,A 180.000,B 0.000,C 180.000} C_DIS
LIN {X 84.420,Y 50.406,Z 73.446,A 180.000,B 0.000,C 180.000} C_DIS
LIN {X 84.467,Y 50.556,Z 73.443,A 180.000,B 0.000,C 180.000} C_DIS
LIN {X 84.513,Y 50.707,Z 73.439,A 180.000,B 0.000,C 180.000} C_DIS
LIN {X 84.559,Y 50.858,Z 73.436,A 180.000,B 0.000,C 180.000} C_DIS
LIN {X 84.606,Y 51.008,Z 73.432,A 180.000,B 0.000,C 180.000} C_DIS
LIN {X 84.652,Y 51.159,Z 73.428,A 180.000,B 0.000,C 180.000} C_DIS
LIN {X 84.698,Y 51.310,Z 73.425,A 180.000,B 0.000,C 180.000} C_DIS
LIN {X 84.744,Y 51.460,Z 73.421,A 180.000,B 0.000,C 180.000} C_DIS
LIN {X 84.790,Y 51.611,Z 73.417,A 180.000,B 0.000,C 180.000} C_DIS
LIN {X 84.835,Y 51.762,Z 73.413,A 180.000,B 0.000,C 180.000} C_DIS
LIN {X 84.881,Y 51.913,Z 73.409,A 180.000,B 0.000,C 180.000} C_DIS
LIN {X 84.927,Y 52.063,Z 73.405,A 180.000,B 0.000,C 180.000} C_DIS
LIN {X 84.972,Y 52.214,Z 73.400,A 180.000,B 0.000,C 180.000} C_DIS
LIN {X 85.017,Y 52.365,Z 73.396,A 180.000,B 0.000,C 180.000} C_DIS
LIN {X 85.063,Y 52.516,Z 73.392,A 180.000,B 0.000,C 180.000} C_DIS
LIN {X 85.108,Y 52.667,Z 73.387,A 180.000,B 0.000,C 180.000} C_DIS
LIN {X 85.153,Y 52.818,Z 73.383,A 180.000,B 0.000,C 180.000} C_DIS
LIN {X 85.198,Y 52.969,Z 73.378,A 180.000,B 0.000,C 180.000} C_DIS
LIN {X 85.243,Y 53.120,Z 73.373,A 180.000,B 0.000,C 180.000} C_DIS
LIN {X 85.288,Y 53.271,Z 73.369,A 180.000,B 0.000,C 180.000} C_DIS
LIN {X 85.333,Y 53.422,Z 73.364,A 180.000,B 0.000,C 180.000} C_DIS
LIN {X 85.378,Y 53.573,Z 73.359,A 180.000,B 0.000,C 180.000} C_DIS
LIN {X 85.422,Y 53.725,Z 73.354,A 180.000,B 0.000,C 180.000} C_DIS
LIN {X 85.445,Y 53.800,Z 73.351,A 180.000,B 0.000,C 180.000} C_DIS
LIN {X 85.467,Y 53.876,Z 73.349,A 180.000,B 0.000,C 180.000} C_DIS
LIN {X 85.489,Y 53.951,Z 73.346,A 180.000,B 0.000,C 180.000} C_DIS
LIN {X 85.511,Y 54.027,Z 73.344,A 180.000,B 0.000,C 180.000} C_DIS
LIN {X 85.534,Y 54.103,Z 73.341,A 180.000,B 0.000,C 180.000} C_DIS
LIN {X 85.556,Y 54.178,Z 73.339,A 180.000,B 0.000,C 180.000} C_DIS
LIN {X 85.578,Y 54.254,Z 73.336,A 180.000,B 0.000,C 180.000} C_DIS
LIN {X 85.600,Y 54.329,Z 73.333,A 180.000,B 0.000,C 180.000} C_DIS
LIN {X 85.622,Y 54.405,Z 73.331,A 180.000,B 0.000,C 180.000} C_DIS
LIN {X 85.645,Y 54.481,Z 73.328,A 180.000,B 0.000,C 180.000} C_DIS
LIN {X 85.667,Y 54.556,Z 73.325,A 180.000,B 0.000,C 180.000} C_DIS
LIN {X 85.689,Y 54.632,Z 73.323,A 180.000,B 0.000,C 180.000} C_DIS
LIN {X 85.711,Y 54.708,Z 73.320,A 180.000,B 0.000,C 180.000} C_DIS
LIN {X 85.733,Y 54.783,Z 73.317,A 180.000,B 0.000,C 180.000} C_DIS
LIN {X 85.754,Y 54.859,Z 73.315,A 180.000,B 0.000,C 180.000} C_DIS
LIN {X 85.776,Y 54.935,Z 73.312,A 180.000,B 0.000,C 180.000} C_DIS
LIN {X 85.798,Y 55.011,Z 73.309,A 180.000,B 0.000,C 180.000} C_DIS
LIN {X 85.820,Y 55.086,Z 73.307,A 180.000,B 0.000,C 180.000} C_DIS
LIN {X 85.842,Y 55.162,Z 73.304,A 180.000,B 0.000,C 180.000} C_DIS
LIN {X 85.864,Y 55.238,Z 73.301,A 180.000,B 0.000,C 180.000} C_DIS
LIN {X 85.886,Y 55.314,Z 73.298,A 180.000,B 0.000,C 180.000} C_DIS
LIN {X 85.908,Y 55.389,Z 73.295,A 180.000,B 0.000,C 180.000} C_DIS
LIN {X 85.930,Y 55.465,Z 73.293,A 180.000,B 0.000,C 180.000} C_DIS
LIN {X 85.951,Y 55.541,Z 73.290,A 180.000,B 0.000,C 180.000} C_DIS
LIN {X 85.973,Y 55.616,Z 73.287,A 180.000,B 0.000,C 180.000} C_DIS
LIN {X 85.995,Y 55.692,Z 73.284,A 180.000,B 0.000,C 180.000} C_DIS
LIN {X 86.017,Y 55.768,Z 73.282,A 180.000,B 0.000,C 180.000} C_DIS
LIN {X 86.039,Y 55.844,Z 73.279,A 180.000,B 0.000,C 180.000} C_DIS
LIN {X 86.061,Y 55.919,Z 73.276,A 180.000,B 0.000,C 180.000} C_DIS
LIN {X 86.083,Y 55.995,Z 73.273,A 180.000,B 0.000,C 180.000} C_DIS
LIN {X 86.105,Y 56.071,Z 73.271,A 180.000,B 0.000,C 180.000} C_DIS
LIN {X 86.127,Y 56.147,Z 73.268,A 180.000,B 0.000,C 180.000} C_DIS
LIN {X 86.148,Y 56.222,Z 73.265,A 180.000,B 0.000,C 180.000} C_DIS
LIN {X 86.170,Y 56.298,Z 73.262,A 180.000,B 0.000,C 180.000} C_DIS
LIN {X 86.192,Y 56.374,Z 73.260,A 180.000,B 0.000,C 180.000} C_DIS
LIN {X 86.214,Y 56.449,Z 73.257,A 180.000,B 0.000,C 180.000} C_DIS
LIN {X 86.236,Y 56.525,Z 73.254,A 180.000,B 0.000,C 180.000} C_DIS
LIN {X 86.258,Y 56.601,Z 73.251,A 180.000,B 0.000,C 180.000} C_DIS
LIN {X 86.302,Y 56.752,Z 73.246,A 180.000,B 0.000,C 180.000} C_DIS
LIN {X 86.367,Y 56.980,Z 73.238,A 180.000,B 0.000,C 180.000} C_DIS
LIN {X 86.411,Y 57.131,Z 73.232,A 180.000,B 0.000,C 180.000} C_DIS
LIN {X 86.433,Y 57.207,Z 73.229,A 180.000,B 0.000,C 180.000} C_DIS
LIN {X 86.477,Y 57.358,Z 73.224,A 180.000,B 0.000,C 180.000} C_DIS
LIN {X 86.542,Y 57.585,Z 73.216,A 180.000,B 0.000,C 180.000} C_DIS
LIN {X 86.586,Y 57.737,Z 73.210,A 180.000,B 0.000,C 180.000} C_DIS
LIN {X 86.608,Y 57.813,Z 73.207,A 180.000,B 0.000,C 180.000} C_DIS
LIN {X 86.652,Y 57.964,Z 73.202,A 180.000,B 0.000,C 180.000} C_DIS
LIN {X 86.717,Y 58.191,Z 73.194,A 180.000,B 0.000,C 180.000} C_DIS
LIN {X 86.761,Y 58.343,Z 73.188,A 180.000,B 0.000,C 180.000} C_DIS
LIN {X 86.783,Y 58.418,Z 73.185,A 180.000,B 0.000,C 180.000} C_DIS
LIN {X 86.827,Y 58.570,Z 73.180,A 180.000,B 0.000,C 180.000} C_DIS
LIN {X 86.892,Y 58.797,Z 73.172,A 180.000,B 0.000,C 180.000} C_DIS
LIN {X 86.936,Y 58.949,Z 73.166,A 180.000,B 0.000,C 180.000} C_DIS
LIN {X 86.958,Y 59.024,Z 73.163,A 180.000,B 0.000,C 180.000} C_DIS
LIN {X 87.002,Y 59.176,Z 73.158,A 180.000,B 0.000,C 180.000} C_DIS
LIN {X 87.067,Y 59.403,Z 73.150,A 180.000,B 0.000,C 180.000} C_DIS
LIN {X 87.111,Y 59.554,Z 73.144,A 180.000,B 0.000,C 180.000} C_DIS
LIN {X 87.133,Y 59.630,Z 73.141,A 180.000,B 0.000,C 180.000} C_DIS
LIN {X 87.174,Y 59.773,Z 73.136,A 180.000,B 0.000,C 180.000} C_DIS
LIN {X 87.195,Y 59.844,Z 73.134,A 180.000,B 0.000,C 180.000} C_DIS
LIN {X 87.216,Y 59.915,Z 73.131,A 180.000,B 0.000,C 180.000} C_DIS
LIN {X 87.246,Y 60.002,Z 73.128,A 180.000,B 0.000,C 180.000} C_DIS
LIN {X 87.279,Y 60.088,Z 73.125,A 180.000,B 0.000,C 180.000} C_DIS
LIN {X 87.324,Y 60.192,Z 73.121,A 180.000,B 0.000,C 180.000} C_DIS
LIN {X 87.374,Y 60.293,Z 73.117,A 180.000,B 0.000,C 180.000} C_DIS
LIN {X 87.422,Y 60.383,Z 73.113,A 180.000,B 0.000,C 180.000} C_DIS
LIN {X 87.474,Y 60.470,Z 73.110,A 180.000,B 0.000,C 180.000} C_DIS
LIN {X 87.540,Y 60.569,Z 73.105,A 180.000,B 0.000,C 180.000} C_DIS
LIN {X 87.611,Y 60.665,Z 73.101,A 180.000,B 0.000,C 180.000} C_DIS
LIN {X 87.689,Y 60.762,Z 73.097,A 180.000,B 0.000,C 180.000} C_DIS
LIN {X 87.772,Y 60.854,Z 73.093,A 180.000,B 0.000,C 180.000} C_DIS
LIN {X 87.851,Y 60.933,Z 73.089,A 180.000,B 0.000,C 180.000} C_DIS
LIN {X 87.934,Y 61.008,Z 73.085,A 180.000,B 0.000,C 180.000} C_DIS
LIN {X 88.031,Y 61.089,Z 73.080,A 180.000,B 0.000,C 180.000} C_DIS
LIN {X 88.133,Y 61.165,Z 73.076,A 180.000,B 0.000,C 180.000} C_DIS
LIN {X 88.247,Y 61.239,Z 73.071,A 180.000,B 0.000,C 180.000} C_DIS
LIN {X 88.365,Y 61.308,Z 73.066,A 180.000,B 0.000,C 180.000} C_DIS
LIN {X 88.485,Y 61.368,Z 73.062,A 180.000,B 0.000,C 180.000} C_DIS
LIN {X 88.608,Y 61.421,Z 73.057,A 180.000,B 0.000,C 180.000} C_DIS
LIN {X 88.740,Y 61.470,Z 73.052,A 180.000,B 0.000,C 180.000} C_DIS
LIN {X 88.876,Y 61.510,Z 73.047,A 180.000,B 0.000,C 180.000} C_DIS
LIN {X 88.948,Y 61.528,Z 73.045,A 180.000,B 0.000,C 180.000} C_DIS
LIN {X 89.021,Y 61.544,Z 73.042,A 180.000,B 0.000,C 180.000} C_DIS
LIN {X 89.095,Y 61.557,Z 73.039,A 180.000,B 0.000,C 180.000} C_DIS
LIN {X 89.169,Y 61.568,Z 73.037,A 180.000,B 0.000,C 180.000} C_DIS
LIN {X 89.245,Y 61.576,Z 73.034,A 180.000,B 0.000,C 180.000} C_DIS
LIN {X 89.321,Y 61.583,Z 73.031,A 180.000,B 0.000,C 180.000} C_DIS
LIN {X 89.398,Y 61.586,Z 73.029,A 180.000,B 0.000,C 180.000} C_DIS
LIN {X 89.474,Y 61.587,Z 73.026,A 180.000,B 0.000,C 180.000} C_DIS
LIN {X 89.555,Y 61.586,Z 73.023,A 180.000,B 0.000,C 180.000} C_DIS
LIN {X 89.636,Y 61.581,Z 73.020,A 180.000,B 0.000,C 180.000} C_DIS
LIN {X 89.716,Y 61.574,Z 73.018,A 180.000,B 0.000,C 180.000} C_DIS
LIN {X 89.797,Y 61.564,Z 73.015,A 180.000,B 0.000,C 180.000} C_DIS
LIN {X 89.875,Y 61.551,Z 73.012,A 180.000,B 0.000,C 180.000} C_DIS
LIN {X 89.953,Y 61.536,Z 73.009,A 180.000,B 0.000,C 180.000} C_DIS
LIN {X 90.030,Y 61.518,Z 73.006,A 180.000,B 0.000,C 180.000} C_DIS
LIN {X 90.107,Y 61.497,Z 73.004,A 180.000,B 0.000,C 180.000} C_DIS
LIN {X 90.182,Y 61.474,Z 73.001,A 180.000,B 0.000,C 180.000} C_DIS
LIN {X 90.257,Y 61.449,Z 72.998,A 180.000,B 0.000,C 180.000} C_DIS
LIN {X 92.719,Y 60.618,Z 72.907,A 180.000,B 0.000,C 180.000} C_DIS
LIN {X 92.943,Y 60.543,Z 72.899,A 180.000,B 0.000,C 180.000} C_DIS
LIN {X 93.689,Y 60.291,Z 72.872,A 180.000,B 0.000,C 180.000} C_DIS
LIN {X 93.913,Y 60.215,Z 72.863,A 180.000,B 0.000,C 180.000} C_DIS
LIN {X 94.062,Y 60.165,Z 72.858,A 180.000,B 0.000,C 180.000} C_DIS
LIN {X 94.510,Y 60.014,Z 72.841,A 180.000,B 0.000,C 180.000} C_DIS
LIN {X 94.659,Y 59.964,Z 72.836,A 180.000,B 0.000,C 180.000} C_DIS
LIN {X 94.808,Y 59.913,Z 72.830,A 180.000,B 0.000,C 180.000} C_DIS
LIN {X 94.883,Y 59.888,Z 72.828,A 180.000,B 0.000,C 180.000} C_DIS
LIN {X 95.032,Y 59.838,Z 72.822,A 180.000,B 0.000,C 180.000} C_DIS
LIN {X 95.107,Y 59.812,Z 72.819,A 180.000,B 0.000,C 180.000} C_DIS
LIN {X 95.180,Y 59.785,Z 72.817,A 180.000,B 0.000,C 180.000} C_DIS
LIN {X 95.254,Y 59.755,Z 72.814,A 180.000,B 0.000,C 180.000} C_DIS
LIN {X 95.327,Y 59.724,Z 72.811,A 180.000,B 0.000,C 180.000} C_DIS
LIN {X 95.398,Y 59.690,Z 72.808,A 180.000,B 0.000,C 180.000} C_DIS
LIN {X 95.469,Y 59.655,Z 72.806,A 180.000,B 0.000,C 180.000} C_DIS
LIN {X 95.540,Y 59.617,Z 72.803,A 180.000,B 0.000,C 180.000} C_DIS
LIN {X 95.610,Y 59.577,Z 72.800,A 180.000,B 0.000,C 180.000} C_DIS
LIN {X 95.678,Y 59.536,Z 72.797,A 180.000,B 0.000,C 180.000} C_DIS
LIN {X 95.746,Y 59.492,Z 72.795,A 180.000,B 0.000,C 180.000} C_DIS
LIN {X 95.809,Y 59.449,Z 72.792,A 180.000,B 0.000,C 180.000} C_DIS
LIN {X 95.871,Y 59.404,Z 72.789,A 180.000,B 0.000,C 180.000} C_DIS
LIN {X 95.932,Y 59.358,Z 72.786,A 180.000,B 0.000,C 180.000} C_DIS
LIN {X 95.991,Y 59.310,Z 72.784,A 180.000,B 0.000,C 180.000} C_DIS
LIN {X 96.048,Y 59.262,Z 72.781,A 180.000,B 0.000,C 180.000} C_DIS
LIN {X 96.104,Y 59.212,Z 72.779,A 180.000,B 0.000,C 180.000} C_DIS
LIN {X 96.158,Y 59.161,Z 72.776,A 180.000,B 0.000,C 180.000} C_DIS
LIN {X 96.210,Y 59.109,Z 72.773,A 180.000,B 0.000,C 180.000} C_DIS
LIN {X 96.308,Y 59.004,Z 72.769,A 180.000,B 0.000,C 180.000} C_DIS
LIN {X 96.401,Y 58.894,Z 72.764,A 180.000,B 0.000,C 180.000} C_DIS
LIN {X 96.485,Y 58.784,Z 72.759,A 180.000,B 0.000,C 180.000} C_DIS
LIN {X 96.564,Y 58.669,Z 72.755,A 180.000,B 0.000,C 180.000} C_DIS
LIN {X 96.636,Y 58.552,Z 72.750,A 180.000,B 0.000,C 180.000} C_DIS
LIN {X 96.702,Y 58.431,Z 72.745,A 180.000,B 0.000,C 180.000} C_DIS
LIN {X 96.760,Y 58.312,Z 72.741,A 180.000,B 0.000,C 180.000} C_DIS
LIN {X 96.812,Y 58.191,Z 72.737,A 180.000,B 0.000,C 180.000} C_DIS
LIN {X 96.858,Y 58.068,Z 72.733,A 180.000,B 0.000,C 180.000} C_DIS
LIN {X 96.898,Y 57.943,Z 72.729,A 180.000,B 0.000,C 180.000} C_DIS
LIN {X 96.932,Y 57.816,Z 72.724,A 180.000,B 0.000,C 180.000} C_DIS
LIN {X 96.960,Y 57.687,Z 72.720,A 180.000,B 0.000,C 180.000} C_DIS
LIN {X 96.980,Y 57.559,Z 72.716,A 180.000,B 0.000,C 180.000} C_DIS
LIN {X 96.995,Y 57.431,Z 72.712,A 180.000,B 0.000,C 180.000} C_DIS
LIN {X 97.003,Y 57.303,Z 72.707,A 180.000,B 0.000,C 180.000} C_DIS
LIN {X 97.005,Y 57.174,Z 72.703,A 180.000,B 0.000,C 180.000} C_DIS
LIN {X 97.001,Y 57.044,Z 72.699,A 180.000,B 0.000,C 180.000} C_DIS
LIN {X 96.990,Y 56.916,Z 72.695,A 180.000,B 0.000,C 180.000} C_DIS
LIN {X 96.971,Y 56.784,Z 72.691,A 180.000,B 0.000,C 180.000} C_DIS
LIN {X 96.946,Y 56.653,Z 72.687,A 180.000,B 0.000,C 180.000} C_DIS
LIN {X 96.912,Y 56.511,Z 72.682,A 180.000,B 0.000,C 180.000} C_DIS
LIN {X 96.876,Y 56.369,Z 72.677,A 180.000,B 0.000,C 180.000} C_DIS
LIN {X 96.856,Y 56.293,Z 72.674,A 180.000,B 0.000,C 180.000} C_DIS
LIN {X 96.837,Y 56.216,Z 72.672,A 180.000,B 0.000,C 180.000} C_DIS
LIN {X 96.817,Y 56.140,Z 72.669,A 180.000,B 0.000,C 180.000} C_DIS
LIN {X 96.798,Y 56.063,Z 72.667,A 180.000,B 0.000,C 180.000} C_DIS
LIN {X 96.778,Y 55.987,Z 72.664,A 180.000,B 0.000,C 180.000} C_DIS
LIN {X 96.759,Y 55.910,Z 72.661,A 180.000,B 0.000,C 180.000} C_DIS
LIN {X 96.739,Y 55.834,Z 72.659,A 180.000,B 0.000,C 180.000} C_DIS
LIN {X 96.719,Y 55.757,Z 72.656,A 180.000,B 0.000,C 180.000} C_DIS
LIN {X 96.700,Y 55.681,Z 72.654,A 180.000,B 0.000,C 180.000} C_DIS
LIN {X 96.680,Y 55.604,Z 72.651,A 180.000,B 0.000,C 180.000} C_DIS
LIN {X 96.660,Y 55.528,Z 72.649,A 180.000,B 0.000,C 180.000} C_DIS
LIN {X 96.641,Y 55.451,Z 72.646,A 180.000,B 0.000,C 180.000} C_DIS
LIN {X 96.601,Y 55.298,Z 72.641,A 180.000,B 0.000,C 180.000} C_DIS
LIN {X 96.561,Y 55.146,Z 72.636,A 180.000,B 0.000,C 180.000} C_DIS
LIN {X 96.521,Y 54.993,Z 72.631,A 180.000,B 0.000,C 180.000} C_DIS
LIN {X 96.481,Y 54.840,Z 72.627,A 180.000,B 0.000,C 180.000} C_DIS
LIN {X 96.441,Y 54.688,Z 72.622,A 180.000,B 0.000,C 180.000} C_DIS
LIN {X 96.400,Y 54.535,Z 72.617,A 180.000,B 0.000,C 180.000} C_DIS
LIN {X 96.360,Y 54.382,Z 72.613,A 180.000,B 0.000,C 180.000} C_DIS
LIN {X 96.319,Y 54.230,Z 72.608,A 180.000,B 0.000,C 180.000} C_DIS
LIN {X 96.278,Y 54.078,Z 72.604,A 180.000,B 0.000,C 180.000} C_DIS
LIN {X 96.237,Y 53.925,Z 72.600,A 180.000,B 0.000,C 180.000} C_DIS
LIN {X 96.196,Y 53.773,Z 72.595,A 180.000,B 0.000,C 180.000} C_DIS
LIN {X 96.155,Y 53.621,Z 72.591,A 180.000,B 0.000,C 180.000} C_DIS
LIN {X 96.113,Y 53.468,Z 72.587,A 180.000,B 0.000,C 180.000} C_DIS
LIN {X 96.072,Y 53.316,Z 72.583,A 180.000,B 0.000,C 180.000} C_DIS
LIN {X 96.030,Y 53.164,Z 72.579,A 180.000,B 0.000,C 180.000} C_DIS
LIN {X 95.988,Y 53.012,Z 72.575,A 180.000,B 0.000,C 180.000} C_DIS
LIN {X 95.946,Y 52.860,Z 72.572,A 180.000,B 0.000,C 180.000} C_DIS
LIN {X 95.903,Y 52.708,Z 72.568,A 180.000,B 0.000,C 180.000} C_DIS
LIN {X 95.861,Y 52.556,Z 72.564,A 180.000,B 0.000,C 180.000} C_DIS
LIN {X 95.818,Y 52.404,Z 72.561,A 180.000,B 0.000,C 180.000} C_DIS
LIN {X 95.775,Y 52.253,Z 72.557,A 180.000,B 0.000,C 180.000} C_DIS
LIN {X 95.732,Y 52.101,Z 72.554,A 180.000,B 0.000,C 180.000} C_DIS
LIN {X 95.688,Y 51.949,Z 72.551,A 180.000,B 0.000,C 180.000} C_DIS
LIN {X 95.645,Y 51.798,Z 72.547,A 180.000,B 0.000,C 180.000} C_DIS
LIN {X 95.601,Y 51.646,Z 72.544,A 180.000,B 0.000,C 180.000} C_DIS
LIN {X 95.557,Y 51.495,Z 72.541,A 180.000,B 0.000,C 180.000} C_DIS
LIN {X 95.513,Y 51.344,Z 72.539,A 180.000,B 0.000,C 180.000} C_DIS
LIN {X 95.469,Y 51.192,Z 72.536,A 180.000,B 0.000,C 180.000} C_DIS
LIN {X 95.424,Y 51.041,Z 72.533,A 180.000,B 0.000,C 180.000} C_DIS
LIN {X 95.380,Y 50.890,Z 72.530,A 180.000,B 0.000,C 180.000} C_DIS
LIN {X 95.289,Y 50.588,Z 72.526,A 180.000,B 0.000,C 180.000} C_DIS
LIN {X 95.199,Y 50.286,Z 72.521,A 180.000,B 0.000,C 180.000} C_DIS
LIN {X 95.107,Y 49.985,Z 72.517,A 180.000,B 0.000,C 180.000} C_DIS
LIN {X 95.014,Y 49.684,Z 72.513,A 180.000,B 0.000,C 180.000} C_DIS
LIN {X 94.920,Y 49.383,Z 72.510,A 180.000,B 0.000,C 180.000} C_DIS
LIN {X 94.826,Y 49.082,Z 72.507,A 180.000,B 0.000,C 180.000} C_DIS
LIN {X 94.730,Y 48.782,Z 72.505,A 180.000,B 0.000,C 180.000} C_DIS
LIN {X 94.633,Y 48.482,Z 72.503,A 180.000,B 0.000,C 180.000} C_DIS
LIN {X 94.536,Y 48.183,Z 72.502,A 180.000,B 0.000,C 180.000} C_DIS
LIN {X 94.437,Y 47.884,Z 72.501,A 180.000,B 0.000,C 180.000} C_DIS
LIN {X 94.338,Y 47.585,Z 72.500,A 180.000,B 0.000,C 180.000} C_DIS
LIN {X 94.288,Y 47.438,Z 72.500,A 180.000,B 0.000,C 180.000} C_DIS
; Cutting Move Starts
LIN {X 90.951,Y 37.545,Z 72.500,A 180.000,B 0.000,C 180.000} C_DIS
LIN {X 90.888,Y 37.366,Z 72.500,A 180.000,B 0.000,C 180.000} C_DIS
LIN {X 90.818,Y 37.206,Z 72.500,A 180.000,B 0.000,C 180.000} C_DIS
LIN {X 90.810,Y 37.187,Z 72.500,A 180.000,B 0.000,C 180.000} C_DIS
LIN {X 90.714,Y 37.009,Z 72.500,A 180.000,B 0.000,C 180.000} C_DIS
LIN {X 90.640,Y 36.890,Z 72.500,A 180.000,B 0.000,C 180.000} C_DIS
LIN {X 90.598,Y 36.830,Z 72.500,A 180.000,B 0.000,C 180.000} C_DIS
LIN {X 90.461,Y 36.653,Z 72.500,A 180.000,B 0.000,C 180.000} C_DIS
LIN {X 90.459,Y 36.651,Z 72.500,A 180.000,B 0.000,C 180.000} C_DIS
LIN {X 90.290,Y 36.472,Z 72.500,A 180.000,B 0.000,C 180.000} C_DIS
LIN {X 90.282,Y 36.465,Z 72.500,A 180.000,B 0.000,C 180.000} C_DIS
LIN {X 90.103,Y 36.310,Z 72.500,A 180.000,B 0.000,C 180.000} C_DIS
LIN {X 90.082,Y 36.294,Z 72.500,A 180.000,B 0.000,C 180.000} C_DIS
LIN {X 89.925,Y 36.182,Z 72.500,A 180.000,B 0.000,C 180.000} C_DIS
LIN {X 89.816,Y 36.115,Z 72.500,A 180.000,B 0.000,C 180.000} C_DIS
LIN {X 89.746,Y 36.075,Z 72.500,A 180.000,B 0.000,C 180.000} C_DIS
LIN {X 89.567,Y 35.988,Z 72.500,A 180.000,B 0.000,C 180.000} C_DIS
LIN {X 89.439,Y 35.936,Z 72.500,A 180.000,B 0.000,C 180.000} C_DIS
LIN {X 89.388,Y 35.917,Z 72.500,A 180.000,B 0.000,C 180.000} C_DIS
LIN {X 89.209,Y 35.862,Z 72.500,A 180.000,B 0.000,C 180.000} C_DIS
LIN {X 89.031,Y 35.821,Z 72.500,A 180.000,B 0.000,C 180.000} C_DIS
LIN {X 88.852,Y 35.793,Z 72.500,A 180.000,B 0.000,C 180.000} C_DIS
LIN {X 88.763,Y 35.784,Z 72.500,A 180.000,B 0.000,C 180.000} C_DIS
LIN {X 88.673,Y 35.778,Z 72.500,A 180.000,B 0.000,C 180.000} C_DIS
LIN {X 88.584,Y 35.776,Z 72.500,A 180.000,B 0.000,C 180.000} C_DIS
LIN {X 88.494,Y 35.777,Z 72.500,A 180.000,B 0.000,C 180.000} C_DIS
LIN {X 88.405,Y 35.781,Z 72.500,A 180.000,B 0.000,C 180.000} C_DIS
LIN {X 88.316,Y 35.788,Z 72.500,A 180.000,B 0.000,C 180.000} C_DIS
LIN {X 88.226,Y 35.798,Z 72.500,A 180.000,B 0.000,C 180.000} C_DIS
LIN {X 88.137,Y 35.812,Z 72.500,A 180.000,B 0.000,C 180.000} C_DIS
LIN {X 88.047,Y 35.829,Z 72.500,A 180.000,B 0.000,C 180.000} C_DIS
LIN {X 87.958,Y 35.849,Z 72.500,A 180.000,B 0.000,C 180.000} C_DIS
LIN {X 87.913,Y 35.861,Z 72.500,A 180.000,B 0.000,C 180.000} C_DIS
LIN {X 87.869,Y 35.873,Z 72.500,A 180.000,B 0.000,C 180.000} C_DIS
LIN {X 87.824,Y 35.886,Z 72.500,A 180.000,B 0.000,C 180.000} C_DIS
LIN {X 87.779,Y 35.901,Z 72.500,A 180.000,B 0.000,C 180.000} C_DIS
LIN {X 87.674,Y 35.936,Z 72.500,A 180.000,B 0.000,C 180.000} C_DIS
LIN {X 81.701,Y 37.951,Z 72.500,A 180.000,B 0.000,C 180.000} C_DIS
LIN {X 81.522,Y 38.012,Z 72.500,A 180.000,B 0.000,C 180.000} C_DIS
LIN {X 81.436,Y 38.045,Z 72.500,A 180.000,B 0.000,C 180.000} C_DIS
LIN {X 81.350,Y 38.081,Z 72.500,A 180.000,B 0.000,C 180.000} C_DIS
LIN {X 81.344,Y 38.084,Z 72.500,A 180.000,B 0.000,C 180.000} C_DIS
LIN {X 81.254,Y 38.126,Z 72.500,A 180.000,B 0.000,C 180.000} C_DIS
LIN {X 81.165,Y 38.173,Z 72.500,A 180.000,B 0.000,C 180.000} C_DIS
LIN {X 81.092,Y 38.215,Z 72.500,A 180.000,B 0.000,C 180.000} C_DIS
LIN {X 81.019,Y 38.260,Z 72.500,A 180.000,B 0.000,C 180.000} C_DIS
LIN {X 80.986,Y 38.281,Z 72.500,A 180.000,B 0.000,C 180.000} C_DIS
LIN {X 80.897,Y 38.343,Z 72.500,A 180.000,B 0.000,C 180.000} C_DIS
LIN {X 80.807,Y 38.412,Z 72.500,A 180.000,B 0.000,C 180.000} C_DIS
LIN {X 80.774,Y 38.439,Z 72.500,A 180.000,B 0.000,C 180.000} C_DIS
LIN {X 80.701,Y 38.501,Z 72.500,A 180.000,B 0.000,C 180.000} C_DIS
LIN {X 80.628,Y 38.569,Z 72.500,A 180.000,B 0.000,C 180.000} C_DIS
LIN {X 80.580,Y 38.618,Z 72.500,A 180.000,B 0.000,C 180.000} C_DIS
LIN {X 80.512,Y 38.690,Z 72.500,A 180.000,B 0.000,C 180.000} C_DIS
LIN {X 80.450,Y 38.762,Z 72.500,A 180.000,B 0.000,C 180.000} C_DIS
LIN {X 80.421,Y 38.796,Z 72.500,A 180.000,B 0.000,C 180.000} C_DIS
LIN {X 80.353,Y 38.886,Z 72.500,A 180.000,B 0.000,C 180.000} C_DIS
LIN {X 80.290,Y 38.975,Z 72.500,A 180.000,B 0.000,C 180.000} C_DIS
LIN {X 80.271,Y 39.004,Z 72.500,A 180.000,B 0.000,C 180.000} C_DIS
LIN {X 80.181,Y 39.154,Z 72.500,A 180.000,B 0.000,C 180.000} C_DIS
LIN {X 80.092,Y 39.331,Z 72.500,A 180.000,B 0.000,C 180.000} C_DIS
LIN {X 80.091,Y 39.333,Z 72.500,A 180.000,B 0.000,C 180.000} C_DIS
LIN {X 80.019,Y 39.511,Z 72.500,A 180.000,B 0.000,C 180.000} C_DIS
LIN {X 79.961,Y 39.690,Z 72.500,A 180.000,B 0.000,C 180.000} C_DIS
LIN {X 79.918,Y 39.869,Z 72.500,A 180.000,B 0.000,C 180.000} C_DIS
LIN {X 79.913,Y 39.893,Z 72.500,A 180.000,B 0.000,C 180.000} C_DIS
LIN {X 79.889,Y 40.048,Z 72.500,A 180.000,B 0.000,C 180.000} C_DIS
LIN {X 79.872,Y 40.226,Z 72.500,A 180.000,B 0.000,C 180.000} C_DIS
LIN {X 79.869,Y 40.405,Z 72.500,A 180.000,B 0.000,C 180.000} C_DIS
LIN {X 79.878,Y 40.584,Z 72.500,A 180.000,B 0.000,C 180.000} C_DIS
LIN {X 79.901,Y 40.763,Z 72.500,A 180.000,B 0.000,C 180.000} C_DIS
LIN {X 79.913,Y 40.835,Z 72.500,A 180.000,B 0.000,C 180.000} C_DIS
LIN {X 79.936,Y 40.942,Z 72.500,A 180.000,B 0.000,C 180.000} C_DIS
LIN {X 79.986,Y 41.120,Z 72.500,A 180.000,B 0.000,C 180.000} C_DIS
LIN {X 80.046,Y 41.299,Z 72.500,A 180.000,B 0.000,C 180.000} C_DIS
LIN {X 86.378,Y 60.070,Z 72.500,A 180.000,B 0.000,C 180.000} C_DIS
LIN {X 86.443,Y 60.249,Z 72.500,A 180.000,B 0.000,C 180.000} C_DIS
LIN {X 86.523,Y 60.427,Z 72.500,A 180.000,B 0.000,C 180.000} C_DIS
LIN {X 86.528,Y 60.437,Z 72.500,A 180.000,B 0.000,C 180.000} C_DIS
LIN {X 86.621,Y 60.606,Z 72.500,A 180.000,B 0.000,C 180.000} C_DIS
LIN {X 86.707,Y 60.739,Z 72.500,A 180.000,B 0.000,C 180.000} C_DIS
LIN {X 86.740,Y 60.785,Z 72.500,A 180.000,B 0.000,C 180.000} C_DIS
LIN {X 86.883,Y 60.964,Z 72.500,A 180.000,B 0.000,C 180.000} C_DIS
LIN {X 86.885,Y 60.967,Z 72.500,A 180.000,B 0.000,C 180.000} C_DIS
LIN {X 87.056,Y 61.143,Z 72.500,A 180.000,B 0.000,C 180.000} C_DIS
LIN {X 87.064,Y 61.150,Z 72.500,A 180.000,B 0.000,C 180.000} C_DIS
LIN {X 87.243,Y 61.301,Z 72.500,A 180.000,B 0.000,C 180.000} C_DIS
LIN {X 87.270,Y 61.321,Z 72.500,A 180.000,B 0.000,C 180.000} C_DIS
LIN {X 87.422,Y 61.425,Z 72.500,A 180.000,B 0.000,C 180.000} C_DIS
LIN {X 87.547,Y 61.500,Z 72.500,A 180.000,B 0.000,C 180.000} C_DIS
LIN {X 87.601,Y 61.529,Z 72.500,A 180.000,B 0.000,C 180.000} C_DIS
LIN {X 87.779,Y 61.614,Z 72.500,A 180.000,B 0.000,C 180.000} C_DIS
LIN {X 87.948,Y 61.679,Z 72.500,A 180.000,B 0.000,C 180.000} C_DIS
LIN {X 87.958,Y 61.682,Z 72.500,A 180.000,B 0.000,C 180.000} C_DIS
LIN {X 88.137,Y 61.735,Z 72.500,A 180.000,B 0.000,C 180.000} C_DIS
LIN {X 88.316,Y 61.775,Z 72.500,A 180.000,B 0.000,C 180.000} C_DIS
LIN {X 88.405,Y 61.789,Z 72.500,A 180.000,B 0.000,C 180.000} C_DIS
LIN {X 88.494,Y 61.800,Z 72.500,A 180.000,B 0.000,C 180.000} C_DIS
LIN {X 88.584,Y 61.808,Z 72.500,A 180.000,B 0.000,C 180.000} C_DIS
LIN {X 88.673,Y 61.813,Z 72.500,A 180.000,B 0.000,C 180.000} C_DIS
LIN {X 88.763,Y 61.815,Z 72.500,A 180.000,B 0.000,C 180.000} C_DIS
LIN {X 88.852,Y 61.813,Z 72.500,A 180.000,B 0.000,C 180.000} C_DIS
LIN {X 88.941,Y 61.808,Z 72.500,A 180.000,B 0.000,C 180.000} C_DIS
LIN {X 89.031,Y 61.800,Z 72.500,A 180.000,B 0.000,C 180.000} C_DIS
LIN {X 89.120,Y 61.789,Z 72.500,A 180.000,B 0.000,C 180.000} C_DIS
LIN {X 89.209,Y 61.774,Z 72.500,A 180.000,B 0.000,C 180.000} C_DIS
LIN {X 89.299,Y 61.756,Z 72.500,A 180.000,B 0.000,C 180.000} C_DIS
LIN {X 89.388,Y 61.735,Z 72.500,A 180.000,B 0.000,C 180.000} C_DIS
LIN {X 89.478,Y 61.710,Z 72.500,A 180.000,B 0.000,C 180.000} C_DIS
LIN {X 89.567,Y 61.682,Z 72.500,A 180.000,B 0.000,C 180.000} C_DIS
LIN {X 95.645,Y 59.631,Z 72.500,A 180.000,B 0.000,C 180.000} C_DIS
LIN {X 95.824,Y 59.570,Z 72.500,A 180.000,B 0.000,C 180.000} C_DIS
LIN {X 95.869,Y 59.552,Z 72.500,A 180.000,B 0.000,C 180.000} C_DIS
LIN {X 95.915,Y 59.534,Z 72.500,A 180.000,B 0.000,C 180.000} C_DIS
LIN {X 95.959,Y 59.515,Z 72.500,A 180.000,B 0.000,C 180.000} C_DIS
LIN {X 96.003,Y 59.495,Z 72.500,A 180.000,B 0.000,C 180.000} C_DIS
LIN {X 96.047,Y 59.474,Z 72.500,A 180.000,B 0.000,C 180.000} C_DIS
LIN {X 96.092,Y 59.451,Z 72.500,A 180.000,B 0.000,C 180.000} C_DIS
LIN {X 96.137,Y 59.428,Z 72.500,A 180.000,B 0.000,C 180.000} C_DIS
LIN {X 96.181,Y 59.403,Z 72.500,A 180.000,B 0.000,C 180.000} C_DIS
LIN {X 96.264,Y 59.355,Z 72.500,A 180.000,B 0.000,C 180.000} C_DIS
LIN {X 96.360,Y 59.292,Z 72.500,A 180.000,B 0.000,C 180.000} C_DIS
LIN {X 96.439,Y 59.236,Z 72.500,A 180.000,B 0.000,C 180.000} C_DIS
LIN {X 96.517,Y 59.176,Z 72.500,A 180.000,B 0.000,C 180.000} C_DIS
LIN {X 96.539,Y 59.158,Z 72.500,A 180.000,B 0.000,C 180.000} C_DIS
LIN {X 96.628,Y 59.082,Z 72.500,A 180.000,B 0.000,C 180.000} C_DIS
LIN {X 96.717,Y 58.997,Z 72.500,A 180.000,B 0.000,C 180.000} C_DIS
LIN {X 96.718,Y 58.996,Z 72.500,A 180.000,B 0.000,C 180.000} C_DIS
LIN {X 96.803,Y 58.907,Z 72.500,A 180.000,B 0.000,C 180.000} C_DIS
LIN {X 96.880,Y 58.819,Z 72.500,A 180.000,B 0.000,C 180.000} C_DIS
LIN {X 96.897,Y 58.798,Z 72.500,A 180.000,B 0.000,C 180.000} C_DIS
LIN {X 97.014,Y 58.640,Z 72.500,A 180.000,B 0.000,C 180.000} C_DIS
LIN {X 97.075,Y 58.546,Z 72.500,A 180.000,B 0.000,C 180.000} C_DIS
LIN {X 97.126,Y 58.461,Z 72.500,A 180.000,B 0.000,C 180.000} C_DIS
LIN {X 97.218,Y 58.282,Z 72.500,A 180.000,B 0.000,C 180.000} C_DIS
LIN {X 97.254,Y 58.201,Z 72.500,A 180.000,B 0.000,C 180.000} C_DIS
LIN {X 97.293,Y 58.103,Z 72.500,A 180.000,B 0.000,C 180.000} C_DIS
LIN {X 97.352,Y 57.925,Z 72.500,A 180.000,B 0.000,C 180.000} C_DIS
LIN {X 97.397,Y 57.746,Z 72.500,A 180.000,B 0.000,C 180.000} C_DIS
LIN {X 97.429,Y 57.567,Z 72.500,A 180.000,B 0.000,C 180.000} C_DIS
LIN {X 97.433,Y 57.535,Z 72.500,A 180.000,B 0.000,C 180.000} C_DIS
LIN {X 97.447,Y 57.388,Z 72.500,A 180.000,B 0.000,C 180.000} C_DIS
LIN {X 97.452,Y 57.210,Z 72.500,A 180.000,B 0.000,C 180.000} C_DIS
LIN {X 97.444,Y 57.031,Z 72.500,A 180.000,B 0.000,C 180.000} C_DIS
LIN {X 97.433,Y 56.918,Z 72.500,A 180.000,B 0.000,C 180.000} C_DIS
LIN {X 97.424,Y 56.852,Z 72.500,A 180.000,B 0.000,C 180.000} C_DIS
LIN {X 97.390,Y 56.673,Z 72.500,A 180.000,B 0.000,C 180.000} C_DIS
LIN {X 97.342,Y 56.495,Z 72.500,A 180.000,B 0.000,C 180.000} C_DIS
LIN {X 97.283,Y 56.316,Z 72.500,A 180.000,B 0.000,C 180.000} C_DIS
LIN {X 94.288,Y 47.438,Z 72.500,A 180.000,B 0.000,C 180.000} C_DIS
; Link Move Starts
LIN {X 94.188,Y 47.139,Z 72.500,A 180.000,B 0.000,C 180.000} C_DIS
LIN {X 94.089,Y 46.840,Z 72.499,A 180.000,B 0.000,C 180.000} C_DIS
LIN {X 93.991,Y 46.541,Z 72.498,A 180.000,B 0.000,C 180.000} C_DIS
LIN {X 93.894,Y 46.241,Z 72.496,A 180.000,B 0.000,C 180.000} C_DIS
LIN {X 93.798,Y 45.941,Z 72.494,A 180.000,B 0.000,C 180.000} C_DIS
LIN {X 93.703,Y 45.641,Z 72.491,A 180.000,B 0.000,C 180.000} C_DIS
LIN {X 93.609,Y 45.340,Z 72.488,A 180.000,B 0.000,C 180.000} C_DIS
LIN {X 93.515,Y 45.039,Z 72.485,A 180.000,B 0.000,C 180.000} C_DIS
LIN {X 93.423,Y 44.738,Z 72.481,A 180.000,B 0.000,C 180.000} C_DIS
LIN {X 93.332,Y 44.436,Z 72.477,A 180.000,B 0.000,C 180.000} C_DIS
LIN {X 93.241,Y 44.135,Z 72.472,A 180.000,B 0.000,C 180.000} C_DIS
LIN {X 93.196,Y 43.984,Z 72.469,A 180.000,B 0.000,C 180.000} C_DIS
LIN {X 93.151,Y 43.832,Z 72.467,A 180.000,B 0.000,C 180.000} C_DIS
LIN {X 93.107,Y 43.681,Z 72.464,A 180.000,B 0.000,C 180.000} C_DIS
LIN {X 93.063,Y 43.530,Z 72.461,A 180.000,B 0.000,C 180.000} C_DIS
LIN {X 93.018,Y 43.379,Z 72.459,A 180.000,B 0.000,C 180.000} C_DIS
LIN {X 92.975,Y 43.227,Z 72.456,A 180.000,B 0.000,C 180.000} C_DIS
LIN {X 92.931,Y 43.076,Z 72.452,A 180.000,B 0.000,C 180.000} C_DIS
LIN {X 92.887,Y 42.924,Z 72.449,A 180.000,B 0.000,C 180.000} C_DIS
LIN {X 92.844,Y 42.773,Z 72.446,A 180.000,B 0.000,C 180.000} C_DIS
LIN {X 92.801,Y 42.621,Z 72.443,A 180.000,B 0.000,C 180.000} C_DIS
LIN {X 92.758,Y 42.469,Z 72.439,A 180.000,B 0.000,C 180.000} C_DIS
LIN {X 92.715,Y 42.317,Z 72.436,A 180.000,B 0.000,C 180.000} C_DIS
LIN {X 92.673,Y 42.165,Z 72.432,A 180.000,B 0.000,C 180.000} C_DIS
LIN {X 92.630,Y 42.014,Z 72.428,A 180.000,B 0.000,C 180.000} C_DIS
LIN {X 92.588,Y 41.862,Z 72.425,A 180.000,B 0.000,C 180.000} C_DIS
LIN {X 92.546,Y 41.710,Z 72.421,A 180.000,B 0.000,C 180.000} C_DIS
LIN {X 92.504,Y 41.557,Z 72.417,A 180.000,B 0.000,C 180.000} C_DIS
LIN {X 92.462,Y 41.405,Z 72.413,A 180.000,B 0.000,C 180.000} C_DIS
LIN {X 92.421,Y 41.253,Z 72.409,A 180.000,B 0.000,C 180.000} C_DIS
LIN {X 92.380,Y 41.101,Z 72.405,A 180.000,B 0.000,C 180.000} C_DIS
LIN {X 92.338,Y 40.948,Z 72.400,A 180.000,B 0.000,C 180.000} C_DIS
LIN {X 92.297,Y 40.796,Z 72.396,A 180.000,B 0.000,C 180.000} C_DIS
LIN {X 92.257,Y 40.644,Z 72.392,A 180.000,B 0.000,C 180.000} C_DIS
LIN {X 92.216,Y 40.491,Z 72.387,A 180.000,B 0.000,C 180.000} C_DIS
LIN {X 92.175,Y 40.339,Z 72.383,A 180.000,B 0.000,C 180.000} C_DIS
LIN {X 92.135,Y 40.186,Z 72.378,A 180.000,B 0.000,C 180.000} C_DIS
LIN {X 92.095,Y 40.033,Z 72.373,A 180.000,B 0.000,C 180.000} C_DIS
LIN {X 92.055,Y 39.881,Z 72.369,A 180.000,B 0.000,C 180.000} C_DIS
LIN {X 92.015,Y 39.728,Z 72.364,A 180.000,B 0.000,C 180.000} C_DIS
LIN {X 91.975,Y 39.575,Z 72.359,A 180.000,B 0.000,C 180.000} C_DIS
LIN {X 91.935,Y 39.422,Z 72.354,A 180.000,B 0.000,C 180.000} C_DIS
LIN {X 91.916,Y 39.346,Z 72.351,A 180.000,B 0.000,C 180.000} C_DIS
LIN {X 91.896,Y 39.269,Z 72.349,A 180.000,B 0.000,C 180.000} C_DIS
LIN {X 91.876,Y 39.193,Z 72.346,A 180.000,B 0.000,C 180.000} C_DIS
LIN {X 91.856,Y 39.116,Z 72.344,A 180.000,B 0.000,C 180.000} C_DIS
LIN {X 91.837,Y 39.040,Z 72.341,A 180.000,B 0.000,C 180.000} C_DIS
LIN {X 91.817,Y 38.963,Z 72.339,A 180.000,B 0.000,C 180.000} C_DIS
LIN {X 91.798,Y 38.887,Z 72.336,A 180.000,B 0.000,C 180.000} C_DIS
LIN {X 91.778,Y 38.810,Z 72.333,A 180.000,B 0.000,C 180.000} C_DIS
LIN {X 91.759,Y 38.734,Z 72.331,A 180.000,B 0.000,C 180.000} C_DIS
LIN {X 91.739,Y 38.657,Z 72.328,A 180.000,B 0.000,C 180.000} C_DIS
LIN {X 91.720,Y 38.581,Z 72.325,A 180.000,B 0.000,C 180.000} C_DIS
LIN {X 91.700,Y 38.504,Z 72.323,A 180.000,B 0.000,C 180.000} C_DIS
LIN {X 91.681,Y 38.428,Z 72.320,A 180.000,B 0.000,C 180.000} C_DIS
LIN {X 91.661,Y 38.351,Z 72.317,A 180.000,B 0.000,C 180.000} C_DIS
LIN {X 91.642,Y 38.275,Z 72.315,A 180.000,B 0.000,C 180.000} C_DIS
LIN {X 91.623,Y 38.198,Z 72.312,A 180.000,B 0.000,C 180.000} C_DIS
LIN {X 91.604,Y 38.121,Z 72.309,A 180.000,B 0.000,C 180.000} C_DIS
LIN {X 91.584,Y 38.045,Z 72.307,A 180.000,B 0.000,C 180.000} C_DIS
LIN {X 91.565,Y 37.968,Z 72.304,A 180.000,B 0.000,C 180.000} C_DIS
LIN {X 91.546,Y 37.891,Z 72.301,A 180.000,B 0.000,C 180.000} C_DIS
LIN {X 91.527,Y 37.815,Z 72.298,A 180.000,B 0.000,C 180.000} C_DIS
LIN {X 91.507,Y 37.738,Z 72.295,A 180.000,B 0.000,C 180.000} C_DIS
LIN {X 91.488,Y 37.662,Z 72.293,A 180.000,B 0.000,C 180.000} C_DIS
LIN {X 91.469,Y 37.585,Z 72.290,A 180.000,B 0.000,C 180.000} C_DIS
LIN {X 91.450,Y 37.509,Z 72.287,A 180.000,B 0.000,C 180.000} C_DIS
LIN {X 91.431,Y 37.432,Z 72.284,A 180.000,B 0.000,C 180.000} C_DIS
LIN {X 91.412,Y 37.359,Z 72.282,A 180.000,B 0.000,C 180.000} C_DIS
LIN {X 91.394,Y 37.286,Z 72.279,A 180.000,B 0.000,C 180.000} C_DIS
LIN {X 91.373,Y 37.214,Z 72.277,A 180.000,B 0.000,C 180.000} C_DIS
LIN {X 91.351,Y 37.142,Z 72.274,A 180.000,B 0.000,C 180.000} C_DIS
LIN {X 91.303,Y 37.013,Z 72.270,A 180.000,B 0.000,C 180.000} C_DIS
LIN {X 91.248,Y 36.888,Z 72.265,A 180.000,B 0.000,C 180.000} C_DIS
LIN {X 91.183,Y 36.756,Z 72.261,A 180.000,B 0.000,C 180.000} C_DIS
LIN {X 91.109,Y 36.629,Z 72.256,A 180.000,B 0.000,C 180.000} C_DIS
LIN {X 91.030,Y 36.511,Z 72.251,A 180.000,B 0.000,C 180.000} C_DIS
LIN {X 90.944,Y 36.398,Z 72.247,A 180.000,B 0.000,C 180.000} C_DIS
LIN {X 90.897,Y 36.340,Z 72.244,A 180.000,B 0.000,C 180.000} C_DIS
LIN {X 90.847,Y 36.284,Z 72.241,A 180.000,B 0.000,C 180.000} C_DIS
LIN {X 90.796,Y 36.229,Z 72.239,A 180.000,B 0.000,C 180.000} C_DIS
LIN {X 90.743,Y 36.176,Z 72.236,A 180.000,B 0.000,C 180.000} C_DIS
LIN {X 90.634,Y 36.077,Z 72.231,A 180.000,B 0.000,C 180.000} C_DIS
LIN {X 90.518,Y 35.985,Z 72.227,A 180.000,B 0.000,C 180.000} C_DIS
LIN {X 90.457,Y 35.941,Z 72.224,A 180.000,B 0.000,C 180.000} C_DIS
LIN {X 90.393,Y 35.898,Z 72.221,A 180.000,B 0.000,C 180.000} C_DIS
LIN {X 90.329,Y 35.858,Z 72.219,A 180.000,B 0.000,C 180.000} C_DIS
LIN {X 90.262,Y 35.819,Z 72.216,A 180.000,B 0.000,C 180.000} C_DIS
LIN {X 90.195,Y 35.784,Z 72.213,A 180.000,B 0.000,C 180.000} C_DIS
LIN {X 90.126,Y 35.750,Z 72.211,A 180.000,B 0.000,C 180.000} C_DIS
LIN {X 90.057,Y 35.719,Z 72.208,A 180.000,B 0.000,C 180.000} C_DIS
LIN {X 89.986,Y 35.690,Z 72.205,A 180.000,B 0.000,C 180.000} C_DIS
LIN {X 89.914,Y 35.663,Z 72.203,A 180.000,B 0.000,C 180.000} C_DIS
LIN {X 89.841,Y 35.639,Z 72.200,A 180.000,B 0.000,C 180.000} C_DIS
LIN {X 89.767,Y 35.618,Z 72.197,A 180.000,B 0.000,C 180.000} C_DIS
LIN {X 89.692,Y 35.599,Z 72.194,A 180.000,B 0.000,C 180.000} C_DIS
LIN {X 89.616,Y 35.582,Z 72.192,A 180.000,B 0.000,C 180.000} C_DIS
LIN {X 89.539,Y 35.569,Z 72.189,A 180.000,B 0.000,C 180.000} C_DIS
LIN {X 89.462,Y 35.558,Z 72.186,A 180.000,B 0.000,C 180.000} C_DIS
LIN {X 89.384,Y 35.550,Z 72.184,A 180.000,B 0.000,C 180.000} C_DIS
LIN {X 89.306,Y 35.544,Z 72.181,A 180.000,B 0.000,C 180.000} C_DIS
LIN {X 89.227,Y 35.542,Z 72.178,A 180.000,B 0.000,C 180.000} C_DIS
LIN {X 89.149,Y 35.542,Z 72.175,A 180.000,B 0.000,C 180.000} C_DIS
LIN {X 89.071,Y 35.545,Z 72.173,A 180.000,B 0.000,C 180.000} C_DIS
LIN {X 88.992,Y 35.551,Z 72.170,A 180.000,B 0.000,C 180.000} C_DIS
LIN {X 88.914,Y 35.560,Z 72.167,A 180.000,B 0.000,C 180.000} C_DIS
LIN {X 88.837,Y 35.572,Z 72.164,A 180.000,B 0.000,C 180.000} C_DIS
LIN {X 88.759,Y 35.586,Z 72.162,A 180.000,B 0.000,C 180.000} C_DIS
LIN {X 88.682,Y 35.604,Z 72.159,A 180.000,B 0.000,C 180.000} C_DIS
LIN {X 88.606,Y 35.624,Z 72.156,A 180.000,B 0.000,C 180.000} C_DIS
LIN {X 88.587,Y 35.629,Z 72.155,A 180.000,B 0.000,C 180.000} C_DIS
LIN {X 88.569,Y 35.635,Z 72.155,A 180.000,B 0.000,C 180.000} C_DIS
LIN {X 88.531,Y 35.647,Z 72.153,A 180.000,B 0.000,C 180.000} C_DIS
LIN {X 88.456,Y 35.672,Z 72.151,A 180.000,B 0.000,C 180.000} C_DIS
LIN {X 88.233,Y 35.748,Z 72.142,A 180.000,B 0.000,C 180.000} C_DIS
LIN {X 88.083,Y 35.798,Z 72.137,A 180.000,B 0.000,C 180.000} C_DIS
LIN {X 87.636,Y 35.949,Z 72.120,A 180.000,B 0.000,C 180.000} C_DIS
LIN {X 87.486,Y 35.999,Z 72.115,A 180.000,B 0.000,C 180.000} C_DIS
LIN {X 87.039,Y 36.150,Z 72.098,A 180.000,B 0.000,C 180.000} C_DIS
LIN {X 86.815,Y 36.226,Z 72.090,A 180.000,B 0.000,C 180.000} C_DIS
LIN {X 85.770,Y 36.578,Z 72.052,A 180.000,B 0.000,C 180.000} C_DIS
LIN {X 85.248,Y 36.754,Z 72.032,A 180.000,B 0.000,C 180.000} C_DIS
LIN {X 84.427,Y 37.031,Z 72.002,A 180.000,B 0.000,C 180.000} C_DIS
LIN {X 80.696,Y 38.290,Z 71.865,A 180.000,B 0.000,C 180.000} C_DIS
LIN {X 80.621,Y 38.315,Z 71.862,A 180.000,B 0.000,C 180.000} C_DIS
LIN {X 80.547,Y 38.343,Z 71.859,A 180.000,B 0.000,C 180.000} C_DIS
LIN {X 80.474,Y 38.372,Z 71.856,A 180.000,B 0.000,C 180.000} C_DIS
LIN {X 80.402,Y 38.403,Z 71.854,A 180.000,B 0.000,C 180.000} C_DIS
LIN {X 80.330,Y 38.437,Z 71.851,A 180.000,B 0.000,C 180.000} C_DIS
LIN {X 80.258,Y 38.473,Z 71.848,A 180.000,B 0.000,C 180.000} C_DIS
LIN {X 80.188,Y 38.510,Z 71.845,A 180.000,B 0.000,C 180.000} C_DIS
LIN {X 80.119,Y 38.550,Z 71.843,A 180.000,B 0.000,C 180.000} C_DIS
LIN {X 80.053,Y 38.591,Z 71.840,A 180.000,B 0.000,C 180.000} C_DIS
LIN {X 79.987,Y 38.633,Z 71.837,A 180.000,B 0.000,C 180.000} C_DIS
LIN {X 79.923,Y 38.678,Z 71.834,A 180.000,B 0.000,C 180.000} C_DIS
LIN {X 79.860,Y 38.724,Z 71.832,A 180.000,B 0.000,C 180.000} C_DIS
LIN {X 79.801,Y 38.770,Z 71.829,A 180.000,B 0.000,C 180.000} C_DIS
LIN {X 79.744,Y 38.817,Z 71.826,A 180.000,B 0.000,C 180.000} C_DIS
LIN {X 79.687,Y 38.866,Z 71.824,A 180.000,B 0.000,C 180.000} C_DIS
LIN {X 79.632,Y 38.916,Z 71.821,A 180.000,B 0.000,C 180.000} C_DIS
LIN {X 79.579,Y 38.967,Z 71.819,A 180.000,B 0.000,C 180.000} C_DIS
LIN {X 79.528,Y 39.020,Z 71.816,A 180.000,B 0.000,C 180.000} C_DIS
LIN {X 79.478,Y 39.073,Z 71.814,A 180.000,B 0.000,C 180.000} C_DIS
LIN {X 79.429,Y 39.128,Z 71.811,A 180.000,B 0.000,C 180.000} C_DIS
LIN {X 79.383,Y 39.183,Z 71.809,A 180.000,B 0.000,C 180.000} C_DIS
LIN {X 79.339,Y 39.239,Z 71.806,A 180.000,B 0.000,C 180.000} C_DIS
LIN {X 79.254,Y 39.355,Z 71.801,A 180.000,B 0.000,C 180.000} C_DIS
LIN {X 79.178,Y 39.471,Z 71.796,A 180.000,B 0.000,C 180.000} C_DIS
LIN {X 79.107,Y 39.591,Z 71.791,A 180.000,B 0.000,C 180.000} C_DIS
LIN {X 79.043,Y 39.714,Z 71.786,A 180.000,B 0.000,C 180.000} C_DIS
LIN {X 78.986,Y 39.841,Z 71.782,A 180.000,B 0.000,C 180.000} C_DIS
LIN {X 78.937,Y 39.964,Z 71.777,A 180.000,B 0.000,C 180.000} C_DIS
LIN {X 78.894,Y 40.089,Z 71.772,A 180.000,B 0.000,C 180.000} C_DIS
LIN {X 78.858,Y 40.215,Z 71.768,A 180.000,B 0.000,C 180.000} C_DIS
LIN {X 78.828,Y 40.343,Z 71.763,A 180.000,B 0.000,C 180.000} C_DIS
LIN {X 78.804,Y 40.477,Z 71.758,A 180.000,B 0.000,C 180.000} C_DIS
LIN {X 78.787,Y 40.612,Z 71.754,A 180.000,B 0.000,C 180.000} C_DIS
LIN {X 78.777,Y 40.744,Z 71.749,A 180.000,B 0.000,C 180.000} C_DIS
LIN {X 78.774,Y 40.877,Z 71.744,A 180.000,B 0.000,C 180.000} C_DIS
LIN {X 78.777,Y 41.005,Z 71.740,A 180.000,B 0.000,C 180.000} C_DIS
LIN {X 78.787,Y 41.133,Z 71.736,A 180.000,B 0.000,C 180.000} C_DIS
LIN {X 78.804,Y 41.266,Z 71.731,A 180.000,B 0.000,C 180.000} C_DIS
LIN {X 78.828,Y 41.397,Z 71.726,A 180.000,B 0.000,C 180.000} C_DIS
LIN {X 78.844,Y 41.467,Z 71.724,A 180.000,B 0.000,C 180.000} C_DIS
LIN {X 78.862,Y 41.537,Z 71.721,A 180.000,B 0.000,C 180.000} C_DIS
LIN {X 78.880,Y 41.607,Z 71.719,A 180.000,B 0.000,C 180.000} C_DIS
LIN {X 78.899,Y 41.676,Z 71.716,A 180.000,B 0.000,C 180.000} C_DIS
LIN {X 78.920,Y 41.752,Z 71.713,A 180.000,B 0.000,C 180.000} C_DIS
LIN {X 78.940,Y 41.828,Z 71.711,A 180.000,B 0.000,C 180.000} C_DIS
LIN {X 78.961,Y 41.905,Z 71.708,A 180.000,B 0.000,C 180.000} C_DIS
LIN {X 78.982,Y 41.981,Z 71.705,A 180.000,B 0.000,C 180.000} C_DIS
LIN {X 79.002,Y 42.057,Z 71.702,A 180.000,B 0.000,C 180.000} C_DIS
LIN {X 79.023,Y 42.133,Z 71.700,A 180.000,B 0.000,C 180.000} C_DIS
